C05472=1215.611,355.008,-74.397,-175.998,7.617,148.292
C05473=1215.607,355.256,-74.430,-175.997,7.621,148.293
C05474=1215.602,355.504,-74.463,-175.995,7.623,148.293
C05475=1215.599,355.752,-74.495,-175.993,7.626,148.293
C05476=1215.595,356.000,-74.528,-175.991,7.629,148.294
C05477=1215.590,356.248,-74.561,-175.990,7.632,148.294
C05478=1215.586,356.496,-74.594,-175.988,7.635,148.294
C05479=1215.582,356.743,-74.625,-175.986,7.638,148.294
C05480=1215.578,356.991,-74.658,-175.985,7.641,148.295
C05481=1215.573,357.239,-74.691,-175.983,7.644,148.295
C05482=1215.569,357.487,-74.724,-175.981,7.646,148.295
C05483=1215.566,357.734,-74.757,-175.979,7.649,148.295
C05484=1215.561,357.982,-74.789,-175.978,7.653,148.296
C05485=1215.557,358.230,-74.822,-175.976,7.655,148.296
C05486=1215.553,358.478,-74.855,-175.974,7.659,148.296
C05487=1215.549,358.726,-74.888,-175.973,7.661,148.297
C05488=1215.545,358.974,-74.920,-175.971,7.664,148.297
C05489=1215.541,359.221,-74.954,-175.969,7.667,148.297
C05490=1215.537,359.469,-74.987,-175.968,7.670,148.297
C05491=1215.533,359.718,-75.019,-175.966,7.673,148.298
C05492=1215.528,359.965,-75.052,-175.964,7.676,148.298
C05493=1215.524,360.212,-75.085,-175.963,7.679,148.298
C05494=1215.520,360.460,-75.118,-175.961,7.681,148.299
C05495=1215.516,360.708,-75.150,-175.959,7.685,148.299
C05496=1215.512,360.956,-75.183,-175.958,7.688,148.299
C05497=1215.508,361.203,-75.216,-175.956,7.690,148.299
C05498=1215.503,361.451,-75.250,-175.954,7.694,148.300
C05499=1215.499,361.699,-75.283,-175.953,7.696,148.300
C05500=1215.495,361.947,-75.316,-175.951,7.699,148.300
C05501=1215.491,362.195,-75.348,-175.950,7.703,148.301
C05502=1215.487,362.443,-75.381,-175.948,7.705,148.301
C05503=1215.482,362.690,-75.415,-175.947,7.708,148.301
C05504=1215.479,362.938,-75.447,-175.945,7.711,148.301
C05505=1215.475,363.186,-75.480,-175.943,7.714,148.302
C05506=1215.471,363.433,-75.513,-175.942,7.717,148.302
C05507=1215.467,363.681,-75.547,-175.941,7.719,148.302
C05508=1215.463,363.929,-75.580,-175.939,7.723,148.303
C05509=1215.458,364.177,-75.613,-175.937,7.726,148.303
C05510=1215.454,364.424,-75.646,-175.936,7.728,148.303
C05511=1215.450,364.673,-75.679,-175.934,7.732,148.304
C05512=1215.446,364.920,-75.712,-175.933,7.735,148.304
C05513=1215.442,365.168,-75.745,-175.931,7.737,148.304
C05514=1215.437,365.416,-75.778,-175.930,7.740,148.305
C05515=1215.433,365.664,-75.811,-175.928,7.744,148.305
C05516=1215.430,365.912,-75.845,-175.927,7.746,148.305
C05517=1215.426,366.160,-75.878,-175.925,7.749,148.306
C05518=1215.421,366.407,-75.911,-175.924,7.752,148.306
C05519=1215.417,366.687,-75.949,-175.922,7.755,148.306
C05520=1215.412,366.967,-75.986,-175.920,7.759,148.307
C05521=1215.408,367.247,-76.024,-175.919,7.761,148.307
C05522=1215.403,367.527,-76.061,-175.917,7.765,148.308
C05523=1215.398,367.775,-76.095,-175.916,7.768,148.308
C05524=1215.394,368.023,-76.128,-175.914,7.770,148.308
C05525=1215.390,368.270,-76.162,-175.913,7.773,148.309
C05526=1215.386,368.518,-76.195,-175.911,7.777,148.309
C05527=1215.382,368.765,-76.228,-175.910,7.780,148.309
C05528=1215.378,369.013,-76.261,-175.909,7.782,148.310
C05529=1215.374,369.261,-76.294,-175.907,7.785,148.310
C05530=1215.370,369.509,-76.328,-175.906,7.788,148.310
C05531=1215.366,369.757,-76.361,-175.905,7.792,148.311
C05532=1215.362,370.005,-76.394,-175.903,7.794,148.311
C05533=1215.358,370.252,-76.428,-175.902,7.797,148.311
C05534=1215.353,370.500,-76.462,-175.900,7.800,148.312
C05535=1215.349,370.748,-76.495,-175.899,7.803,148.312
C05536=1215.345,370.995,-76.528,-175.898,7.805,148.313
C05537=1215.341,371.243,-76.561,-175.897,7.808,148.313
C05538=1215.337,371.490,-76.595,-175.895,7.812,148.313
C05539=1215.334,371.739,-76.628,-175.894,7.814,148.314
C05540=1215.329,371.987,-76.662,-175.892,7.817,148.314
C05541=1215.325,372.234,-76.695,-175.891,7.820,148.314
C05542=1215.321,372.482,-76.729,-175.890,7.823,148.315
C05543=1215.317,372.729,-76.762,-175.889,7.826,148.315
C05544=1215.312,372.977,-76.796,-175.888,7.828,148.316
C05545=1215.308,373.225,-76.829,-175.886,7.831,148.316
C05546=1215.304,373.473,-76.864,-175.885,7.834,148.316
C05547=1215.300,373.721,-76.897,-175.884,7.837,148.317
C05548=1215.296,373.968,-76.930,-175.883,7.840,148.317
C05549=1215.292,374.215,-76.964,-175.881,7.843,148.318
C05550=1215.288,374.463,-76.997,-175.880,7.846,148.318
C05551=1215.283,374.711,-77.031,-175.879,7.849,148.318
C05552=1215.279,374.958,-77.065,-175.877,7.852,148.319
C05553=1215.276,375.207,-77.098,-175.876,7.855,148.319
C05554=1215.272,375.454,-77.131,-175.875,7.857,148.320
C05555=1215.268,375.702,-77.165,-175.874,7.860,148.320
C05556=1215.263,375.950,-77.199,-175.873,7.863,148.320
C05557=1215.259,376.197,-77.232,-175.872,7.866,148.321
C05558=1215.256,376.445,-77.266,-175.870,7.869,148.321
C05559=1215.252,376.693,-77.299,-175.869,7.871,148.322
C05560=1215.247,376.940,-77.334,-175.868,7.874,148.322
C05561=1215.243,377.188,-77.367,-175.867,7.877,148.322
C05562=1215.239,377.435,-77.401,-175.866,7.880,148.323
C05563=1215.235,377.684,-77.435,-175.864,7.883,148.323
C05564=1215.231,377.932,-77.468,-175.863,7.886,148.323
C05565=1215.227,378.179,-77.502,-175.862,7.888,148.324
C05566=1215.223,378.426,-77.535,-175.861,7.891,148.324
C05567=1215.218,378.674,-77.570,-175.860,7.894,148.325
C05568=1215.215,378.922,-77.603,-175.859,7.896,148.325
C05569=1215.211,379.169,-77.637,-175.858,7.899,148.326
C05570=1215.206,379.417,-77.671,-175.857,7.902,148.326
C05571=1215.202,379.665,-77.705,-175.856,7.905,148.326
C05572=1215.198,379.912,-77.738,-175.855,7.908,148.327
C05573=1215.194,380.160,-77.773,-175.853,7.910,148.327
C05574=1215.190,380.408,-77.806,-175.853,7.913,148.328
C05575=1215.186,380.655,-77.840,-175.852,7.916,148.328
C05576=1215.181,380.903,-77.873,-175.850,7.919,148.329
C05577=1215.178,381.151,-77.908,-175.849,7.922,148.329
C05578=1215.174,381.398,-77.942,-175.848,7.925,148.329
C05579=1215.169,381.646,-77.975,-175.848,7.927,148.330
C05580=1215.165,381.893,-78.009,-175.847,7.930,148.330
C05581=1215.161,382.142,-78.043,-175.845,7.933,148.331
C05582=1215.157,382.389,-78.077,-175.844,7.935,148.331
C05583=1215.153,382.636,-78.111,-175.843,7.939,148.332
C05584=1215.148,382.884,-78.145,-175.842,7.941,148.332
C05585=1215.145,383.132,-78.179,-175.842,7.943,148.332
C05586=1215.140,383.380,-78.213,-175.840,7.946,148.333
C05587=1215.137,383.627,-78.247,-175.840,7.949,148.333
C05588=1215.133,383.875,-78.281,-175.838,7.952,148.334
C05589=1215.128,384.123,-78.315,-175.837,7.955,148.334
C05590=1215.125,384.370,-78.348,-175.837,7.957,148.335
C05591=1215.120,384.618,-78.383,-175.836,7.960,148.335
C05592=1215.116,384.866,-78.416,-175.835,7.963,148.336
C05593=1215.112,385.114,-78.451,-175.834,7.966,148.336
C05594=1215.108,385.361,-78.485,-175.833,7.969,148.337
C05595=1215.105,385.608,-78.519,-175.832,7.971,148.337
C05596=1215.100,385.857,-78.553,-175.831,7.974,148.337
C05597=1215.096,386.104,-78.587,-175.830,7.977,148.338
C05598=1215.092,386.351,-78.621,-175.829,7.979,148.338
C05599=1215.088,386.599,-78.655,-175.828,7.981,148.339
C05600=1215.083,386.847,-78.689,-175.828,7.985,148.339
C05601=1215.080,387.094,-78.723,-175.826,7.987,148.340
C05602=1215.076,387.342,-78.758,-175.826,7.989,148.340
C05603=1215.072,387.590,-78.791,-175.825,7.992,148.340
C05604=1215.067,387.837,-78.825,-175.824,7.995,148.341
C05605=1215.064,388.085,-78.860,-175.824,7.998,148.341
C05606=1215.059,388.332,-78.894,-175.822,8.000,148.342
C05607=1215.055,388.580,-78.928,-175.821,8.003,148.342
C05608=1215.051,388.828,-78.962,-175.821,8.005,148.343
C05609=1215.047,389.075,-78.996,-175.820,8.008,148.343
C05610=1215.043,389.323,-79.030,-175.819,8.011,148.344
C05611=1215.039,389.571,-79.065,-175.818,8.013,148.344
C05612=1215.035,389.818,-79.099,-175.817,8.016,148.344
C05613=1215.031,390.066,-79.132,-175.817,8.019,148.345
C05614=1215.027,390.314,-79.167,-175.816,8.021,148.345
C05615=1215.023,390.561,-79.201,-175.815,8.024,148.346
C05616=1215.018,390.808,-79.235,-175.814,8.027,148.346
C05617=1215.015,391.056,-79.270,-175.814,8.029,148.347
C05618=1215.011,391.304,-79.304,-175.813,8.032,148.347
C05619=1215.007,391.552,-79.339,-175.812,8.035,148.348
C05620=1215.003,391.799,-79.373,-175.811,8.037,148.348
C05621=1214.998,392.047,-79.407,-175.811,8.039,148.349
C05622=1214.995,392.295,-79.441,-175.810,8.042,148.349
C05623=1214.990,392.576,-79.480,-175.809,8.046,148.350
C05624=1214.985,392.859,-79.519,-175.808,8.048,148.350
C05625=1214.981,393.141,-79.558,-175.807,8.051,148.351
C05626=1214.976,393.422,-79.598,-175.806,8.055,148.351
C05627=1214.972,393.670,-79.632,-175.806,8.057,148.352
C05628=1214.968,393.918,-79.666,-175.805,8.060,148.352
C05629=1214.963,394.166,-79.700,-175.804,8.062,148.353
C05630=1214.959,394.414,-79.735,-175.804,8.065,148.353
C05631=1214.956,394.661,-79.769,-175.803,8.067,148.354
C05632=1214.951,394.908,-79.803,-175.802,8.070,148.354
C05633=1214.948,395.156,-79.838,-175.802,8.072,148.355
C05634=1214.943,395.404,-79.872,-175.801,8.075,148.355
C05635=1214.939,395.652,-79.907,-175.800,8.077,148.355
C05636=1214.935,395.899,-79.941,-175.799,8.080,148.356
C05637=1214.931,396.146,-79.975,-175.799,8.082,148.356
C05638=1214.927,396.394,-80.010,-175.799,8.084,148.357
C05639=1214.923,396.641,-80.044,-175.797,8.087,148.357
C05640=1214.919,396.890,-80.079,-175.797,8.089,148.358
C05641=1214.915,397.137,-80.113,-175.796,8.092,148.358
C05642=1214.911,397.383,-80.148,-175.796,8.094,148.359
C05643=1214.907,397.632,-80.183,-175.795,8.097,148.359
C05644=1214.902,397.879,-80.217,-175.794,8.099,148.360
C05645=1214.899,398.127,-80.251,-175.794,8.101,148.360
C05646=1214.895,398.374,-80.286,-175.793,8.105,148.361
C05647=1214.891,398.622,-80.321,-175.792,8.107,148.361
C05648=1214.887,398.869,-80.355,-175.792,8.110,148.362
C05649=1214.882,399.117,-80.389,-175.791,8.112,148.362
C05650=1214.878,399.365,-80.424,-175.791,8.114,148.363
C05651=1214.875,399.612,-80.458,-175.790,8.117,148.363
C05652=1214.871,399.860,-80.493,-175.789,8.119,148.363
C05653=1214.866,400.108,-80.527,-175.789,8.121,148.364
C05654=1214.863,400.355,-80.562,-175.788,8.124,148.364
C05655=1214.858,400.602,-80.596,-175.788,8.126,148.365
C05656=1214.855,400.850,-80.631,-175.787,8.128,148.365
C05657=1214.850,401.098,-80.666,-175.786,8.131,148.366
C05658=1214.846,401.345,-80.700,-175.786,8.134,148.366
C05659=1214.842,401.593,-80.734,-175.785,8.136,148.367
C05660=1214.838,401.840,-80.769,-175.785,8.139,148.367
C05661=1214.834,402.088,-80.804,-175.784,8.141,148.368
C05662=1214.830,402.335,-80.838,-175.784,8.143,148.368
C05663=1214.826,402.583,-80.873,-175.783,8.145,148.369
C05664=1214.822,402.831,-80.908,-175.782,8.148,148.369
C05665=1214.818,403.079,-80.942,-175.782,8.150,148.369
C05666=1214.814,403.326,-80.976,-175.782,8.152,148.370
C05667=1214.810,403.573,-81.012,-175.781,8.155,148.371
C05668=1214.806,403.821,-81.046,-175.780,8.157,148.371
C05669=1214.802,404.069,-81.081,-175.780,8.160,148.371
C05670=1214.798,404.316,-81.115,-175.779,8.162,148.372
C05671=1214.794,404.563,-81.151,-175.779,8.165,148.372
C05672=1214.789,404.811,-81.185,-175.778,8.167,148.373
C05673=1214.786,405.059,-81.220,-175.778,8.169,148.373
C05674=1214.782,405.306,-81.254,-175.778,8.171,148.374
C05675=1214.778,405.554,-81.289,-175.777,8.173,148.374
C05676=1214.773,405.801,-81.324,-175.776,8.176,148.375
C05677=1214.769,406.049,-81.359,-175.775,8.178,148.375
C05678=1214.765,406.297,-81.393,-175.775,8.181,148.376
C05679=1214.762,406.544,-81.428,-175.775,8.183,148.376
C05680=1214.757,406.791,-81.462,-175.774,8.185,148.377
C05681=1214.753,407.039,-81.497,-175.774,8.188,148.377
C05682=1214.749,407.287,-81.532,-175.773,8.190,148.377
C05683=1214.745,407.534,-81.567,-175.773,8.192,148.378
C05684=1214.741,407.782,-81.602,-175.772,8.194,148.378
C05685=1214.737,408.029,-81.636,-175.772,8.196,148.379
C05686=1214.733,408.276,-81.671,-175.771,8.198,148.379
C05687=1214.729,408.524,-81.706,-175.771,8.202,148.380
C05688=1214.725,408.772,-81.741,-175.770,8.204,148.380
C05689=1214.721,409.019,-81.776,-175.770,8.206,148.381
C05690=1214.716,409.267,-81.811,-175.770,8.208,148.381
C05691=1214.713,409.514,-81.845,-175.769,8.210,148.382
C05692=1214.709,409.761,-81.880,-175.769,8.212,148.382
C05693=1214.705,410.009,-81.915,-175.768,8.214,148.382
C05694=1214.701,410.258,-81.950,-175.767,8.217,148.383
C05695=1214.697,410.504,-81.985,-175.767,8.219,148.383
C05696=1214.693,410.752,-82.020,-175.766,8.222,148.384
C05697=1214.689,411.000,-82.054,-175.766,8.224,148.384
C05698=1214.685,411.247,-82.089,-175.766,8.226,148.385
C05699=1214.681,411.494,-82.124,-175.765,8.228,148.385
C05700=1214.677,411.742,-82.159,-175.765,8.230,148.386
C05701=1214.672,411.989,-82.194,-175.764,8.232,148.386
C05702=1214.668,412.238,-82.228,-175.764,8.234,148.386
C05703=1214.664,412.484,-82.264,-175.764,8.237,148.387
C05704=1214.660,412.732,-82.298,-175.763,8.239,148.387
C05705=1214.657,412.980,-82.334,-175.763,8.241,148.388
C05706=1214.653,413.227,-82.368,-175.762,8.244,148.388
C05707=1214.649,413.475,-82.403,-175.761,8.246,148.389
C05708=1214.644,413.722,-82.438,-175.761,8.248,148.389
C05709=1214.641,413.970,-82.473,-175.761,8.250,148.390
C05710=1214.636,414.217,-82.508,-175.760,8.252,148.390
C05711=1214.632,414.465,-82.543,-175.760,8.254,148.391
C05712=1214.629,414.713,-82.578,-175.759,8.257,148.391
C05713=1214.624,414.960,-82.613,-175.759,8.259,148.391
C05714=1214.620,415.207,-82.648,-175.759,8.261,148.392
C05715=1214.616,415.442,-82.681,-175.758,8.263,148.392
C05716=1214.612,415.679,-82.714,-175.758,8.265,148.393
C05717=1214.608,415.914,-82.747,-175.757,8.267,148.393
C05718=1214.605,416.150,-82.781,-175.756,8.269,148.394
C05719=1214.601,416.385,-82.814,-175.757,8.271,148.394
C05720=1214.597,416.620,-82.848,-175.756,8.273,148.394
C05721=1214.595,416.856,-82.880,-175.756,8.275,148.395
C05722=1214.596,417.090,-82.914,-175.755,8.277,148.395
C05723=1214.175,417.091,-82.949,-175.759,8.287,148.399
C05724=1214.174,416.855,-82.917,-175.759,8.285,148.398
C05725=1214.175,416.618,-82.883,-175.759,8.283,148.398
C05726=1214.180,416.381,-82.849,-175.760,8.281,148.398
C05727=1214.183,416.144,-82.816,-175.760,8.280,148.397
C05728=1214.187,415.906,-82.782,-175.760,8.278,148.397
C05729=1214.190,415.671,-82.749,-175.761,8.276,148.396
C05730=1214.194,415.433,-82.715,-175.761,8.274,148.396
C05731=1214.199,415.197,-82.682,-175.761,8.271,148.396
C05732=1214.202,414.949,-82.647,-175.762,8.269,148.395
C05733=1214.206,414.702,-82.612,-175.762,8.267,148.395
C05734=1214.210,414.454,-82.577,-175.763,8.265,148.394
C05735=1214.215,414.207,-82.542,-175.763,8.263,148.394
C05736=1214.219,413.959,-82.507,-175.764,8.261,148.393
C05737=1214.222,413.711,-82.472,-175.764,8.259,148.393
C05738=1214.227,413.464,-82.437,-175.765,8.257,148.393
C05739=1214.230,413.217,-82.402,-175.765,8.254,148.392
C05740=1214.235,412.969,-82.367,-175.765,8.252,148.391
C05741=1214.239,412.721,-82.332,-175.766,8.249,148.391
C05742=1214.243,412.474,-82.297,-175.767,8.247,148.391
C05743=1214.247,412.226,-82.263,-175.767,8.245,148.390
C05744=1214.251,411.980,-82.228,-175.767,8.243,148.390
C05745=1214.255,411.731,-82.193,-175.768,8.241,148.389
C05746=1214.258,411.484,-82.157,-175.768,8.238,148.389
C05747=1214.263,411.237,-82.123,-175.769,8.236,148.388
C05748=1214.267,410.988,-82.088,-175.769,8.234,148.388
C05749=1214.271,410.742,-82.053,-175.769,8.232,148.387
C05750=1214.275,410.493,-82.018,-175.770,8.230,148.387
C05751=1214.279,410.246,-81.984,-175.770,8.228,148.387
C05752=1214.283,409.999,-81.949,-175.771,8.225,148.386
C05753=1214.287,409.751,-81.914,-175.772,8.223,148.386
C05754=1214.291,409.504,-81.879,-175.772,8.221,148.385
C05755=1214.295,409.257,-81.844,-175.772,8.218,148.385
C05756=1214.299,409.008,-81.809,-175.773,8.216,148.384
C05757=1214.303,408.761,-81.774,-175.773,8.214,148.384
C05758=1214.307,408.514,-81.740,-175.774,8.212,148.383
C05759=1214.311,408.266,-81.705,-175.774,8.210,148.383
C05760=1214.315,408.019,-81.670,-175.775,8.207,148.382
C05761=1214.319,407.771,-81.635,-175.776,8.205,148.382
C05762=1214.324,407.523,-81.601,-175.776,8.203,148.382
C05763=1214.327,407.276,-81.565,-175.776,8.200,148.381
C05764=1214.331,407.029,-81.531,-175.777,8.198,148.381
C05765=1214.335,406.781,-81.496,-175.777,8.196,148.380
C05766=1214.340,406.533,-81.462,-175.778,8.193,148.380
C05767=1214.343,406.286,-81.426,-175.778,8.191,148.379
C05768=1214.348,406.038,-81.392,-175.779,8.189,148.379
C05769=1214.351,405.790,-81.358,-175.779,8.187,148.378
C05770=1214.355,405.544,-81.323,-175.779,8.184,148.378
C05771=1214.359,405.296,-81.288,-175.780,8.182,148.377
C05772=1214.364,405.048,-81.253,-175.781,8.179,148.377
C05773=1214.368,404.800,-81.218,-175.781,8.177,148.377
C05774=1214.372,404.554,-81.184,-175.782,8.175,148.376
C05775=1214.375,404.305,-81.149,-175.783,8.172,148.376
C05776=1214.380,404.058,-81.115,-175.783,8.170,148.375
C05777=1214.384,403.810,-81.080,-175.783,8.168,148.374
C05778=1214.388,403.563,-81.046,-175.784,8.166,148.374
C05779=1214.392,403.315,-81.010,-175.785,8.163,148.374
C05780=1214.396,403.068,-80.976,-175.785,8.161,148.373
C05781=1214.400,402.820,-80.941,-175.785,8.158,148.373
C05782=1214.405,402.572,-80.907,-175.786,8.156,148.372
C05783=1214.408,402.324,-80.872,-175.787,8.153,148.372
C05784=1214.412,402.078,-80.837,-175.787,8.151,148.371
C05785=1214.416,401.830,-80.802,-175.788,8.149,148.371
C05786=1214.421,401.582,-80.768,-175.788,8.146,148.370
C05787=1214.424,401.334,-80.734,-175.789,8.144,148.370
C05788=1214.428,401.087,-80.699,-175.789,8.142,148.369
C05789=1214.433,400.840,-80.665,-175.790,8.139,148.369
C05790=1214.436,400.592,-80.630,-175.791,8.137,148.368
C05791=1214.441,400.345,-80.595,-175.791,8.134,148.368
C05792=1214.444,400.097,-80.560,-175.792,8.132,148.368
C05793=1214.449,399.849,-80.526,-175.792,8.129,148.367
C05794=1214.452,399.602,-80.492,-175.793,8.127,148.367
C05795=1214.457,399.354,-80.457,-175.794,8.124,148.366
C05796=1214.461,399.106,-80.422,-175.794,8.122,148.366
C05797=1214.465,398.859,-80.389,-175.795,8.120,148.365
C05798=1214.469,398.612,-80.353,-175.796,8.117,148.365
C05799=1214.473,398.364,-80.318,-175.796,8.115,148.364
C05800=1214.477,398.117,-80.285,-175.796,8.113,148.364
C05801=1214.481,397.869,-80.250,-175.797,8.110,148.363
C05802=1214.485,397.621,-80.215,-175.797,8.108,148.363
C05803=1214.489,397.373,-80.180,-175.799,8.105,148.362
C05804=1214.493,397.126,-80.147,-175.799,8.102,148.362
C05805=1214.498,396.879,-80.112,-175.800,8.100,148.361
C05806=1214.502,396.631,-80.077,-175.800,8.097,148.361
C05807=1214.505,396.383,-80.043,-175.801,8.095,148.361
C05808=1214.509,396.135,-80.009,-175.802,8.092,148.360
C05809=1214.513,395.888,-79.975,-175.802,8.090,148.360
C05810=1214.517,395.640,-79.940,-175.803,8.087,148.359
C05811=1214.522,395.393,-79.905,-175.804,8.085,148.359
C05812=1214.526,395.146,-79.872,-175.804,8.082,148.358
C05813=1214.530,394.897,-79.837,-175.805,8.080,148.358
C05814=1214.534,394.650,-79.802,-175.806,8.077,148.357
C05815=1214.537,394.402,-79.768,-175.806,8.075,148.357
C05816=1214.542,394.155,-79.734,-175.807,8.072,148.356
C05817=1214.546,393.908,-79.700,-175.807,8.070,148.356
C05818=1214.550,393.660,-79.665,-175.809,8.067,148.355
C05819=1214.554,393.412,-79.630,-175.809,8.065,148.355
C05820=1214.558,393.130,-79.591,-175.810,8.062,148.354
C05821=1214.563,392.848,-79.552,-175.811,8.059,148.354
C05822=1214.568,392.566,-79.513,-175.812,8.056,148.353
C05823=1214.573,392.283,-79.474,-175.813,8.053,148.353
C05824=1214.576,392.036,-79.440,-175.813,8.050,148.352
C05825=1214.581,391.789,-79.406,-175.814,8.048,148.352
C05826=1214.584,391.541,-79.371,-175.815,8.045,148.351
C05827=1214.589,391.293,-79.337,-175.816,8.043,148.351
C05828=1214.593,391.046,-79.303,-175.816,8.039,148.350
C05829=1214.597,390.798,-79.268,-175.817,8.038,148.350
C05830=1214.601,390.550,-79.234,-175.818,8.034,148.349
C05831=1214.605,390.302,-79.200,-175.819,8.032,148.349
C05832=1214.609,390.055,-79.166,-175.820,8.030,148.349
C05833=1214.613,389.808,-79.132,-175.820,8.026,148.348
C05834=1214.617,389.560,-79.097,-175.821,8.025,148.348
C05835=1214.621,389.313,-79.063,-175.822,8.021,148.347
C05836=1214.625,389.065,-79.029,-175.823,8.019,148.347
C05837=1214.629,388.817,-78.995,-175.823,8.016,148.346
C05838=1214.633,388.569,-78.961,-175.824,8.014,148.346
C05839=1214.637,388.322,-78.927,-175.825,8.011,148.345
C05840=1214.641,388.074,-78.892,-175.826,8.008,148.345
C05841=1214.645,387.827,-78.858,-175.827,8.006,148.344
C05842=1214.650,387.579,-78.824,-175.828,8.003,148.344
C05843=1214.653,387.331,-78.790,-175.828,8.001,148.344
C05844=1214.658,387.084,-78.756,-175.829,7.998,148.343
C05845=1214.662,386.837,-78.722,-175.830,7.995,148.343
C05846=1214.666,386.588,-78.688,-175.831,7.992,148.342
C05847=1214.670,386.341,-78.654,-175.832,7.990,148.342
C05848=1214.674,386.093,-78.619,-175.833,7.987,148.341
C05849=1214.678,385.846,-78.585,-175.834,7.984,148.341
C05850=1214.682,385.598,-78.551,-175.835,7.981,148.340
C05851=1214.686,385.350,-78.517,-175.835,7.979,148.340
C05852=1214.691,385.103,-78.483,-175.837,7.976,148.339
C05853=1214.694,384.855,-78.449,-175.838,7.973,148.339
C05854=1214.698,384.607,-78.416,-175.838,7.970,148.338
C05855=1214.703,384.360,-78.381,-175.839,7.968,148.338
C05856=1214.706,384.112,-78.347,-175.840,7.965,148.338
C05857=1214.711,383.864,-78.313,-175.841,7.962,148.337
C05858=1214.715,383.617,-78.279,-175.842,7.959,148.337
C05859=1214.719,383.370,-78.245,-175.843,7.957,148.336
C05860=1214.723,383.121,-78.211,-175.844,7.955,148.336
C05861=1214.727,382.874,-78.177,-175.845,7.951,148.335
C05862=1214.732,382.626,-78.144,-175.846,7.949,148.335
C05863=1214.735,382.378,-78.109,-175.847,7.946,148.335
C05864=1214.739,382.131,-78.075,-175.848,7.943,148.334
C05865=1214.743,381.883,-78.042,-175.849,7.940,148.334
C05866=1214.747,381.636,-78.008,-175.850,7.937,148.333
C05867=1214.752,381.387,-77.974,-175.851,7.935,148.333
C05868=1214.755,381.140,-77.940,-175.852,7.932,148.333
C05869=1214.759,380.893,-77.906,-175.853,7.929,148.332
C05870=1214.764,380.645,-77.872,-175.854,7.926,148.332
C05871=1214.767,380.397,-77.838,-175.855,7.924,148.331
C05872=1214.772,380.149,-77.804,-175.856,7.921,148.331
C05873=1214.776,379.902,-77.770,-175.858,7.918,148.330
C05874=1214.780,379.654,-77.737,-175.858,7.915,148.330
C05875=1214.785,379.407,-77.703,-175.860,7.912,148.329
C05876=1214.788,379.158,-77.669,-175.861,7.909,148.329
C05877=1214.792,378.911,-77.635,-175.861,7.907,148.329
C05878=1214.797,378.663,-77.602,-175.863,7.904,148.328
C05879=1214.801,378.416,-77.568,-175.864,7.902,148.328
C05880=1214.804,378.168,-77.534,-175.865,7.899,148.327
C05881=1214.808,377.921,-77.500,-175.866,7.896,148.327
C05882=1214.813,377.673,-77.467,-175.867,7.893,148.326
C05883=1214.817,377.426,-77.433,-175.868,7.890,148.326
C05884=1214.821,377.178,-77.400,-175.869,7.887,148.326
C05885=1214.825,376.930,-77.365,-175.871,7.884,148.325
C05886=1214.829,376.682,-77.332,-175.872,7.882,148.325
C05887=1214.833,376.434,-77.298,-175.873,7.879,148.324
C05888=1214.837,376.187,-77.265,-175.874,7.876,148.324
C05889=1214.842,375.939,-77.231,-175.875,7.873,148.324
C05890=1214.845,375.691,-77.197,-175.876,7.870,148.323
C05891=1214.849,375.444,-77.163,-175.878,7.867,148.323
C05892=1214.853,375.196,-77.130,-175.879,7.865,148.323
C05893=1214.858,374.948,-77.096,-175.880,7.862,148.322
C05894=1214.862,374.701,-77.063,-175.881,7.859,148.322
C05895=1214.866,374.453,-77.030,-175.882,7.856,148.321
C05896=1214.870,374.205,-76.995,-175.884,7.853,148.321
C05897=1214.874,373.957,-76.962,-175.885,7.850,148.320
C05898=1214.879,373.709,-76.928,-175.887,7.847,148.320
C05899=1214.882,373.462,-76.895,-175.888,7.844,148.320
C05900=1214.887,373.215,-76.861,-175.889,7.841,148.319
C05901=1214.891,372.967,-76.828,-175.890,7.839,148.319
C05902=1214.895,372.720,-76.794,-175.891,7.836,148.319
C05903=1214.899,372.471,-76.760,-175.893,7.833,148.318
C05904=1214.903,372.223,-76.727,-175.894,7.830,148.318
C05905=1214.907,371.975,-76.694,-175.895,7.827,148.317
C05906=1214.911,371.728,-76.660,-175.897,7.825,148.317
C05907=1214.915,371.481,-76.627,-175.898,7.821,148.317
C05908=1214.919,371.233,-76.594,-175.900,7.818,148.316
C05909=1214.923,370.985,-76.561,-175.901,7.815,148.316
C05910=1214.927,370.737,-76.526,-175.902,7.813,148.316
C05911=1214.931,370.489,-76.493,-175.903,7.810,148.315
C05912=1214.936,370.242,-76.459,-175.904,7.807,148.315
C05913=1214.940,369.994,-76.426,-175.906,7.804,148.315
C05914=1214.944,369.746,-76.393,-175.908,7.801,148.314
C05915=1214.948,369.498,-76.360,-175.909,7.798,148.314
C05916=1214.952,369.251,-76.326,-175.910,7.795,148.313
C05917=1214.956,369.004,-76.293,-175.911,7.792,148.313
C05918=1214.960,368.756,-76.260,-175.913,7.790,148.313
C05919=1214.965,368.508,-76.226,-175.915,7.786,148.312
C05920=1214.969,368.260,-76.193,-175.916,7.783,148.312
C05921=1214.973,368.012,-76.159,-175.917,7.781,148.312
C05922=1214.977,367.764,-76.126,-175.919,7.778,148.311
C05923=1214.981,367.516,-76.093,-175.920,7.775,148.311
C05924=1214.986,367.237,-76.056,-175.922,7.772,148.311
C05925=1214.990,366.957,-76.018,-175.923,7.768,148.310
C05926=1214.994,366.677,-75.980,-175.925,7.765,148.310
C05927=1215.000,366.396,-75.943,-175.927,7.762,148.309
C05928=1215.004,366.148,-75.910,-175.928,7.759,148.309
C05929=1215.008,365.901,-75.876,-175.930,7.756,148.309
C05930=1215.012,365.653,-75.843,-175.931,7.753,148.308
C05931=1215.016,365.405,-75.810,-175.932,7.750,148.308
C05932=1215.020,365.158,-75.777,-175.934,7.747,148.308
C05933=1215.025,364.910,-75.744,-175.936,7.744,148.307
C05934=1215.029,364.662,-75.711,-175.937,7.741,148.307
C05935=1215.033,364.414,-75.677,-175.939,7.738,148.307
C05936=1215.037,364.167,-75.644,-175.940,7.736,148.306
C05937=1215.040,363.919,-75.612,-175.942,7.732,148.306
C05938=1215.044,363.671,-75.578,-175.943,7.729,148.306
C05939=1215.048,363.423,-75.545,-175.944,7.727,148.305
C05940=1215.052,363.175,-75.512,-175.947,7.723,148.305
C05941=1215.056,362.928,-75.479,-175.948,7.720,148.305
C05942=1215.060,362.680,-75.446,-175.949,7.718,148.305
C05943=1215.065,362.432,-75.412,-175.951,7.715,148.304
C05944=1215.069,362.184,-75.380,-175.953,7.712,148.304
C05945=1215.073,361.936,-75.347,-175.954,7.709,148.304
C05946=1215.077,361.688,-75.314,-175.956,7.706,148.303
C05947=1215.082,361.441,-75.281,-175.957,7.703,148.303
C05948=1215.086,361.194,-75.248,-175.959,7.700,148.303
C05949=1215.090,360.946,-75.215,-175.960,7.697,148.302
C05950=1215.094,360.698,-75.183,-175.962,7.694,148.302
C05951=1215.098,360.450,-75.150,-175.964,7.692,148.302
C05952=1215.102,360.202,-75.116,-175.965,7.689,148.302
C05953=1215.106,359.955,-75.083,-175.967,7.685,148.301
C05954=1215.111,359.707,-75.050,-175.969,7.683,148.301
C05955=1215.115,359.459,-75.018,-175.970,7.680,148.301
C05956=1215.118,359.211,-74.985,-175.973,7.677,148.300
C05957=1215.123,358.963,-74.952,-175.974,7.674,148.300
C05958=1215.127,358.715,-74.919,-175.976,7.671,148.300
C05959=1215.131,358.467,-74.886,-175.977,7.668,148.299
C05960=1215.135,358.220,-74.853,-175.979,7.665,148.299
C05961=1215.139,357.972,-74.820,-175.981,7.662,148.299
C05962=1215.143,357.724,-74.788,-175.982,7.659,148.299
C05963=1215.147,357.476,-74.755,-175.984,7.657,148.298
C05964=1215.151,357.228,-74.722,-175.986,7.653,148.298
C05965=1215.156,356.980,-74.689,-175.987,7.650,148.298
C05966=1215.160,356.733,-74.657,-175.989,7.647,148.298
C05967=1215.164,356.486,-74.624,-175.991,7.644,148.297
C05968=1215.168,356.237,-74.592,-175.992,7.642,148.297
C05969=1215.173,355.989,-74.558,-175.994,7.638,148.297
C05970=1215.176,355.741,-74.527,-175.996,7.636,148.297
C05971=1215.180,355.494,-74.493,-175.998,7.633,148.296
C05972=1215.185,355.246,-74.460,-175.999,7.630,148.296
C05973=1215.189,354.998,-74.428,-176.001,7.627,148.296
C05974=1215.192,354.750,-74.395,-176.003,7.624,148.296
C05975=1215.197,354.503,-74.363,-176.005,7.621,148.295
C05976=1215.202,354.255,-74.330,-176.007,7.619,148.295
C05977=1215.206,354.007,-74.298,-176.008,7.615,148.295
C05978=1215.209,353.759,-74.265,-176.010,7.613,148.295
C05979=1215.214,353.511,-74.233,-176.012,7.609,148.294
C05980=1215.218,353.263,-74.199,-176.014,7.607,148.294
C05981=1215.222,353.016,-74.168,-176.016,7.603,148.294
C05982=1215.226,352.768,-74.135,-176.017,7.601,148.294
C05983=1215.231,352.520,-74.102,-176.019,7.598,148.293
C05984=1215.234,352.272,-74.070,-176.021,7.595,148.293
C05985=1215.239,352.024,-74.037,-176.023,7.592,148.293
C05986=1215.243,351.775,-74.005,-176.025,7.589,148.293
C05987=1215.247,351.529,-73.973,-176.026,7.586,148.293
C05988=1215.252,351.280,-73.940,-176.028,7.584,148.292
C05989=1215.255,351.033,-73.908,-176.030,7.580,148.292
C05990=1215.260,350.785,-73.875,-176.032,7.578,148.292
C05991=1215.264,350.536,-73.843,-176.034,7.574,148.292
C05992=1215.268,350.290,-73.811,-176.035,7.572,148.291
C05993=1215.272,350.041,-73.778,-176.038,7.568,148.291
C05994=1215.276,349.793,-73.746,-176.039,7.566,148.291
C05995=1215.280,349.545,-73.713,-176.041,7.563,148.291
C05996=1215.285,349.297,-73.681,-176.043,7.560,148.291
C05997=1215.289,349.050,-73.649,-176.045,7.557,148.290
C05998=1215.293,348.802,-73.616,-176.047,7.554,148.290
C05999=1215.297,348.554,-73.584,-176.049,7.552,148.290
C06000=1215.301,348.306,-73.552,-176.051,7.548,148.290
C06001=1215.306,348.058,-73.520,-176.052,7.546,148.290
C06002=1215.310,347.811,-73.487,-176.054,7.543,148.289
C06003=1215.313,347.563,-73.455,-176.056,7.540,148.289
C06004=1215.318,347.314,-73.423,-176.058,7.537,148.289
C06005=1215.322,347.067,-73.392,-176.060,7.534,148.289
C06006=1215.326,346.819,-73.358,-176.062,7.531,148.289
C06007=1215.330,346.571,-73.327,-176.064,7.528,148.288
C06008=1215.334,346.323,-73.294,-176.066,7.526,148.288
C06009=1215.339,346.075,-73.263,-176.068,7.522,148.288
C06010=1215.343,345.827,-73.230,-176.069,7.520,148.288
C06011=1215.347,345.579,-73.198,-176.071,7.517,148.288
C06012=1215.351,345.331,-73.165,-176.073,7.514,148.287
C06013=1215.355,345.084,-73.134,-176.075,7.511,148.287
C06014=1215.360,344.836,-73.101,-176.077,7.508,148.287
C06015=1215.364,344.588,-73.069,-176.079,7.505,148.287
C06016=1215.369,344.340,-73.037,-176.081,7.502,148.287
C06017=1215.372,344.092,-73.005,-176.083,7.500,148.286
C06018=1215.376,343.844,-72.974,-176.085,7.496,148.286
C06019=1215.381,343.596,-72.942,-176.087,7.494,148.286
C06020=1215.385,343.348,-72.910,-176.089,7.491,148.286
C06021=1215.389,343.100,-72.877,-176.091,7.488,148.286
C06022=1215.393,342.852,-72.846,-176.092,7.486,148.286
C06023=1215.397,342.604,-72.814,-176.095,7.482,148.285
C06024=1215.402,342.356,-72.781,-176.096,7.480,148.285
C06025=1215.406,342.109,-72.750,-176.099,7.477,148.285
C06026=1215.410,341.860,-72.718,-176.101,7.474,148.285
C06027=1215.414,341.612,-72.686,-176.103,7.471,148.285
C06028=1215.418,341.335,-72.650,-176.105,7.467,148.285
C06029=1215.423,341.057,-72.614,-176.107,7.464,148.284
C06030=1215.428,340.779,-72.579,-176.109,7.462,148.284
C06031=1215.433,340.501,-72.543,-176.111,7.459,148.284
C06032=1215.437,340.253,-72.511,-176.114,7.455,148.284
C06033=1215.441,340.006,-72.479,-176.115,7.453,148.284
C06034=1215.446,339.757,-72.447,-176.117,7.449,148.283
C06035=1215.449,339.509,-72.415,-176.120,7.447,148.284
C06036=1215.454,339.261,-72.384,-176.122,7.444,148.283
C06037=1215.458,339.013,-72.352,-176.123,7.441,148.283
C06038=1215.463,338.766,-72.321,-176.126,7.438,148.283
C06039=1215.466,338.518,-72.289,-176.128,7.436,148.283
C06040=1215.470,338.269,-72.257,-176.130,7.432,148.283
C06041=1215.475,338.022,-72.225,-176.132,7.430,148.283
C06042=1215.479,337.773,-72.194,-176.134,7.427,148.283
C06043=1215.483,337.526,-72.162,-176.136,7.424,148.282
C06044=1215.487,337.278,-72.130,-176.138,7.421,148.282
C06045=1215.492,337.029,-72.098,-176.140,7.418,148.282
C06046=1215.496,336.782,-72.066,-176.142,7.415,148.282
C06047=1215.500,336.533,-72.035,-176.144,7.413,148.282
C06048=1215.504,336.286,-72.004,-176.146,7.409,148.282
C06049=1215.508,336.038,-71.972,-176.148,7.407,148.282
C06050=1215.513,335.790,-71.941,-176.150,7.405,148.281
C06051=1215.517,335.542,-71.909,-176.152,7.401,148.281
C06052=1215.521,335.294,-71.877,-176.154,7.399,148.281
C06053=1215.525,335.046,-71.846,-176.156,7.396,148.281
C06054=1215.529,334.798,-71.814,-176.158,7.393,148.281
C06055=1215.533,334.550,-71.783,-176.161,7.390,148.281
C06056=1215.537,334.302,-71.752,-176.162,7.388,148.281
C06057=1215.542,334.054,-71.720,-176.165,7.385,148.281
C06058=1215.546,333.806,-71.688,-176.167,7.382,148.280
C06059=1215.551,333.558,-71.657,-176.169,7.379,148.280
C06060=1215.554,333.310,-71.625,-176.171,7.377,148.280
C06061=1215.559,333.062,-71.594,-176.173,7.373,148.280
C06062=1215.563,332.814,-71.563,-176.175,7.371,148.280
C06063=1215.567,332.567,-71.531,-176.178,7.368,148.280
C06064=1215.571,332.318,-71.500,-176.179,7.365,148.280
C06065=1215.575,332.071,-71.468,-176.182,7.362,148.280
C06066=1215.579,331.822,-71.437,-176.184,7.360,148.280
C06067=1215.584,331.575,-71.406,-176.186,7.356,148.280
C06068=1215.588,331.326,-71.375,-176.188,7.354,148.279
C06069=1215.593,331.078,-71.343,-176.190,7.351,148.279
C06070=1215.597,330.830,-71.311,-176.192,7.348,148.279
C06071=1215.601,330.582,-71.280,-176.195,7.345,148.279
C06072=1215.606,330.334,-71.249,-176.196,7.343,148.279
C06073=1215.610,330.086,-71.218,-176.199,7.340,148.279
C06074=1215.614,329.838,-71.187,-176.201,7.337,148.279
C06075=1215.618,329.590,-71.156,-176.203,7.334,148.279
C06076=1215.622,329.342,-71.124,-176.205,7.332,148.279
C06077=1215.626,329.094,-71.093,-176.208,7.329,148.279
C06078=1215.631,328.846,-71.062,-176.209,7.326,148.278
C06079=1215.635,328.599,-71.031,-176.212,7.323,148.278
C06080=1215.639,328.350,-71.000,-176.214,7.321,148.278
C06081=1215.643,328.103,-70.969,-176.216,7.318,148.278
C06082=1215.647,327.854,-70.938,-176.218,7.315,148.278
C06083=1215.651,327.606,-70.907,-176.221,7.312,148.278
C06084=1215.655,327.358,-70.876,-176.222,7.309,148.278
C06085=1215.660,327.110,-70.844,-176.225,7.306,148.278
C06086=1215.664,326.862,-70.813,-176.227,7.304,148.278
C06087=1215.668,326.614,-70.782,-176.229,7.301,148.278
C06088=1215.673,326.366,-70.751,-176.231,7.299,148.278
C06089=1215.677,326.118,-70.720,-176.234,7.295,148.278
C06090=1215.681,325.870,-70.689,-176.236,7.293,148.278
C06091=1215.685,325.622,-70.659,-176.238,7.290,148.277
C06092=1215.689,325.374,-70.627,-176.240,7.287,148.277
C06093=1215.694,325.126,-70.596,-176.243,7.284,148.277
C06094=1215.698,324.878,-70.565,-176.244,7.282,148.277
C06095=1215.702,324.629,-70.534,-176.247,7.279,148.277
C06096=1215.707,324.381,-70.503,-176.249,7.276,148.277
C06097=1215.711,324.133,-70.473,-176.251,7.273,148.277
C06098=1215.714,323.886,-70.441,-176.253,7.271,148.277
C06099=1215.719,323.638,-70.411,-176.256,7.268,148.277
C06100=1215.724,323.390,-70.380,-176.258,7.266,148.277
C06101=1215.728,323.141,-70.349,-176.260,7.262,148.277
C06102=1215.732,322.893,-70.318,-176.262,7.260,148.277
C06103=1215.736,322.646,-70.288,-176.265,7.257,148.277
C06104=1215.740,322.397,-70.257,-176.266,7.254,148.277
C06105=1215.745,322.149,-70.226,-176.268,7.252,148.277
C06106=1215.749,321.901,-70.195,-176.271,7.249,148.277
C06107=1215.753,321.653,-70.165,-176.273,7.247,148.277
C06108=1215.757,321.405,-70.133,-176.275,7.244,148.276
C06109=1215.762,321.157,-70.102,-176.278,7.241,148.277
C06110=1215.766,320.909,-70.071,-176.280,7.238,148.277
C06111=1215.769,320.661,-70.041,-176.282,7.236,148.276
C06112=1215.774,320.413,-70.010,-176.285,7.233,148.276
C06113=1215.779,320.165,-69.980,-176.287,7.231,148.276
C06114=1215.782,319.916,-69.950,-176.289,7.227,148.276
C06115=1215.787,319.668,-69.919,-176.291,7.225,148.276
C06116=1215.791,319.420,-69.888,-176.294,7.222,148.276
C06117=1215.795,319.172,-69.858,-176.296,7.220,148.276
C06118=1215.799,318.924,-69.827,-176.298,7.216,148.276
C06119=1215.804,318.676,-69.796,-176.300,7.214,148.276
C06120=1215.808,318.428,-69.766,-176.303,7.211,148.276
C06121=1215.812,318.180,-69.735,-176.305,7.209,148.276
C06122=1215.816,317.932,-69.704,-176.307,7.206,148.276
C06123=1215.820,317.684,-69.674,-176.309,7.203,148.276
C06124=1215.825,317.435,-69.644,-176.312,7.200,148.276
C06125=1215.830,317.188,-69.613,-176.314,7.198,148.276
C06126=1215.833,316.939,-69.583,-176.316,7.195,148.276
C06127=1215.838,316.691,-69.552,-176.318,7.193,148.276
C06128=1215.842,316.444,-69.522,-176.321,7.189,148.276
C06129=1215.847,316.195,-69.492,-176.323,7.187,148.276
C06130=1215.851,315.947,-69.461,-176.326,7.184,148.276
C06131=1215.854,315.699,-69.430,-176.327,7.182,148.276
C06132=1215.859,315.423,-69.396,-176.330,7.179,148.276
C06133=1215.864,315.146,-69.362,-176.333,7.176,148.276
C06134=1215.868,314.871,-69.329,-176.335,7.173,148.276
C06135=1215.874,314.595,-69.296,-176.338,7.170,148.276
C06136=1215.878,314.347,-69.264,-176.340,7.167,148.276
C06137=1215.882,314.099,-69.234,-176.343,7.164,148.276
C06138=1215.887,313.850,-69.204,-176.345,7.162,148.276
C06139=1215.891,313.603,-69.174,-176.347,7.159,148.276
C06140=1215.895,313.355,-69.143,-176.349,7.157,148.276
C06141=1215.899,313.107,-69.114,-176.352,7.153,148.276
C06142=1215.903,312.858,-69.083,-176.354,7.151,148.276
C06143=1215.908,312.610,-69.053,-176.357,7.148,148.276
C06144=1215.912,312.362,-69.023,-176.359,7.146,148.276
C06145=1215.916,312.114,-68.992,-176.361,7.144,148.276
C06146=1215.921,311.865,-68.962,-176.363,7.140,148.276
C06147=1215.925,311.618,-68.932,-176.365,7.138,148.276
C06148=1215.929,311.370,-68.903,-176.368,7.135,148.276
C06149=1215.934,311.122,-68.872,-176.370,7.133,148.276
C06150=1215.937,310.873,-68.842,-176.373,7.130,148.276
C06151=1215.942,310.625,-68.811,-176.375,7.128,148.276
C06152=1215.946,310.376,-68.782,-176.377,7.125,148.276
C06153=1215.951,310.128,-68.751,-176.380,7.122,148.276
C06154=1215.955,309.880,-68.722,-176.382,7.119,148.276
C06155=1215.959,309.632,-68.691,-176.384,7.117,148.276
C06156=1215.964,309.384,-68.661,-176.387,7.114,148.276
C06157=1215.968,309.136,-68.631,-176.389,7.112,148.276
C06158=1215.972,308.888,-68.602,-176.391,7.109,148.276
C06159=1215.976,308.640,-68.571,-176.393,7.106,148.276
C06160=1215.981,308.392,-68.542,-176.396,7.103,148.276
C06161=1215.985,308.143,-68.512,-176.398,7.101,148.276
C06162=1215.989,307.896,-68.481,-176.400,7.099,148.276
C06163=1215.994,307.647,-68.452,-176.403,7.096,148.276
C06164=1215.998,307.399,-68.421,-176.405,7.094,148.276
C06165=1216.002,307.151,-68.392,-176.408,7.091,148.276
C06166=1216.007,306.903,-68.362,-176.410,7.088,148.276
C06167=1216.010,306.654,-68.332,-176.413,7.085,148.276
C06168=1216.015,306.406,-68.302,-176.415,7.083,148.276
C06169=1216.019,306.158,-68.272,-176.417,7.080,148.276
C06170=1216.023,305.910,-68.242,-176.420,7.078,148.276
C06171=1216.028,305.661,-68.212,-176.422,7.075,148.276
C06172=1216.032,305.413,-68.183,-176.424,7.073,148.276
C06173=1216.036,305.165,-68.153,-176.427,7.070,148.276
C06174=1216.040,304.917,-68.123,-176.429,7.067,148.276
C06175=1216.045,304.669,-68.093,-176.431,7.065,148.276
C06176=1216.050,304.421,-68.064,-176.434,7.062,148.276
C06177=1216.054,304.173,-68.034,-176.436,7.060,148.276
C06178=1216.058,303.925,-68.005,-176.439,7.057,148.276
C06179=1216.063,303.677,-67.974,-176.441,7.055,148.277
C06180=1216.067,303.428,-67.945,-176.443,7.052,148.277
C06181=1216.071,303.180,-67.915,-176.446,7.050,148.277
C06182=1216.075,302.932,-67.886,-176.448,7.046,148.277
C06183=1216.079,302.683,-67.856,-176.450,7.044,148.277
C06184=1216.084,302.435,-67.827,-176.452,7.042,148.277
C06185=1216.088,302.187,-67.797,-176.455,7.039,148.277
C06186=1216.092,301.939,-67.767,-176.457,7.037,148.277
C06187=1216.096,301.691,-67.737,-176.460,7.034,148.277
C06188=1216.101,301.442,-67.708,-176.462,7.032,148.277
C06189=1216.105,301.194,-67.678,-176.465,7.029,148.277
C06190=1216.109,300.946,-67.649,-176.467,7.026,148.277
C06191=1216.113,300.698,-67.619,-176.470,7.024,148.277
C06192=1216.117,300.449,-67.590,-176.472,7.021,148.277
C06193=1216.123,300.202,-67.560,-176.474,7.019,148.277
C06194=1216.127,299.953,-67.531,-176.477,7.016,148.277
C06195=1216.131,299.705,-67.501,-176.479,7.014,148.277
C06196=1216.135,299.457,-67.472,-176.482,7.011,148.277
C06197=1216.140,299.208,-67.442,-176.484,7.009,148.277
C06198=1216.144,298.960,-67.413,-176.486,7.006,148.277
C06199=1216.148,298.712,-67.384,-176.489,7.003,148.278
C06200=1216.152,298.464,-67.354,-176.491,7.001,148.278
C06201=1216.156,298.215,-67.325,-176.494,6.999,148.278
C06202=1216.161,297.968,-67.296,-176.496,6.996,148.278
C06203=1216.165,297.720,-67.266,-176.499,6.993,148.278
C06204=1216.170,297.471,-67.237,-176.501,6.991,148.278
C06205=1216.174,297.222,-67.208,-176.503,6.988,148.278
C06206=1216.178,296.974,-67.178,-176.506,6.986,148.278
C06207=1216.182,296.726,-67.149,-176.508,6.984,148.278
C06208=1216.187,296.478,-67.120,-176.510,6.981,148.278
C06209=1216.191,296.230,-67.090,-176.513,6.979,148.278
C06210=1216.196,295.982,-67.061,-176.516,6.976,148.278
C06211=1216.200,295.733,-67.032,-176.518,6.973,148.278
C06212=1216.204,295.485,-67.003,-176.520,6.971,148.279
C06213=1216.208,295.236,-66.973,-176.523,6.968,148.279
C06214=1216.213,294.988,-66.944,-176.525,6.966,148.279
C06215=1216.217,294.740,-66.915,-176.527,6.963,148.279
C06216=1216.222,294.492,-66.886,-176.530,6.961,148.279
C06217=1216.226,294.243,-66.857,-176.533,6.958,148.279
C06218=1216.229,293.995,-66.828,-176.535,6.956,148.279
C06219=1216.235,293.747,-66.799,-176.537,6.954,148.279
C06220=1216.239,293.499,-66.770,-176.540,6.951,148.279
C06221=1216.243,293.251,-66.740,-176.542,6.949,148.279
C06222=1216.247,293.002,-66.711,-176.545,6.946,148.279
C06223=1216.252,292.753,-66.682,-176.547,6.943,148.279
C06224=1216.256,292.506,-66.653,-176.549,6.941,148.279
C06225=1216.261,292.257,-66.624,-176.552,6.938,148.279
C06226=1216.264,292.009,-66.596,-176.554,6.936,148.280
C06227=1216.268,291.761,-66.566,-176.557,6.933,148.280
C06228=1216.274,291.513,-66.538,-176.559,6.931,148.280
C06229=1216.278,291.264,-66.508,-176.561,6.929,148.280
C06230=1216.282,291.016,-66.479,-176.564,6.926,148.280
C06231=1216.286,290.767,-66.450,-176.567,6.924,148.280
C06232=1216.290,290.520,-66.422,-176.569,6.922,148.280
C06233=1216.295,290.271,-66.393,-176.571,6.919,148.280
C06234=1216.299,290.023,-66.363,-176.573,6.917,148.280
C06235=1216.304,289.775,-66.335,-176.577,6.914,148.281
C06236=1216.309,289.501,-66.303,-176.579,6.912,148.281
C06237=1216.314,289.227,-66.271,-176.581,6.909,148.281
C06238=1216.318,288.952,-66.239,-176.585,6.906,148.281
C06239=1216.323,288.678,-66.208,-176.587,6.903,148.281
C06240=1216.327,288.430,-66.178,-176.589,6.901,148.281
C06241=1216.331,288.181,-66.150,-176.592,6.899,148.281
C06242=1216.336,287.933,-66.121,-176.595,6.896,148.281
C06243=1216.340,287.684,-66.092,-176.597,6.893,148.281
C06244=1216.344,287.436,-66.064,-176.599,6.891,148.281
C06245=1216.349,287.188,-66.035,-176.602,6.889,148.282
C06246=1216.353,286.939,-66.006,-176.604,6.886,148.282
C06247=1216.358,286.691,-65.977,-176.607,6.883,148.282
C06248=1216.362,286.443,-65.949,-176.609,6.881,148.282
C06249=1216.366,286.194,-65.920,-176.612,6.879,148.282
C06250=1216.371,285.946,-65.891,-176.614,6.876,148.282
C06251=1216.375,285.698,-65.863,-176.616,6.874,148.282
C06252=1216.379,285.449,-65.834,-176.619,6.872,148.283
C06253=1216.383,285.201,-65.806,-176.622,6.869,148.283
C06254=1216.388,284.953,-65.777,-176.624,6.867,148.283
C06255=1216.392,284.704,-65.748,-176.626,6.865,148.283
C06256=1216.396,284.457,-65.720,-176.629,6.862,148.283
C06257=1216.401,284.208,-65.691,-176.631,6.860,148.283
C06258=1216.405,283.959,-65.663,-176.634,6.857,148.283
C06259=1216.410,283.711,-65.635,-176.636,6.855,148.283
C06260=1216.414,283.463,-65.606,-176.639,6.853,148.283
C06261=1216.418,283.215,-65.578,-176.641,6.850,148.283
C06262=1216.423,282.966,-65.549,-176.644,6.848,148.284
C06263=1216.427,282.719,-65.521,-176.646,6.845,148.284
C06264=1216.432,282.470,-65.492,-176.649,6.842,148.284
C06265=1216.436,282.221,-65.464,-176.651,6.841,148.284
C06266=1216.440,281.974,-65.435,-176.653,6.838,148.284
C06267=1216.445,281.725,-65.406,-176.656,6.835,148.284
C06268=1216.449,281.477,-65.379,-176.659,6.833,148.284
C06269=1216.453,281.228,-65.350,-176.661,6.831,148.285
C06270=1216.458,280.980,-65.322,-176.663,6.828,148.285
C06271=1216.462,280.731,-65.293,-176.666,6.826,148.285
C06272=1216.466,280.483,-65.265,-176.668,6.824,148.285
C06273=1216.471,280.234,-65.237,-176.671,6.821,148.285
C06274=1216.475,279.986,-65.209,-176.673,6.819,148.285
C06275=1216.480,279.738,-65.180,-176.676,6.817,148.285
C06276=1216.483,279.490,-65.151,-176.679,6.814,148.286
C06277=1216.488,279.242,-65.124,-176.681,6.812,148.286
C06278=1216.492,278.993,-65.095,-176.683,6.810,148.286
C06279=1216.497,278.745,-65.067,-176.686,6.807,148.286
C06280=1216.501,278.496,-65.038,-176.688,6.805,148.286
C06281=1216.505,278.248,-65.011,-176.690,6.803,148.286
C06282=1216.510,277.999,-64.982,-176.694,6.800,148.286
C06283=1216.515,277.751,-64.955,-176.696,6.798,148.286
C06284=1216.518,277.502,-64.927,-176.698,6.796,148.287
C06285=1216.523,277.254,-64.898,-176.701,6.793,148.287
C06286=1216.527,277.006,-64.870,-176.703,6.791,148.287
C06287=1216.532,276.758,-64.842,-176.706,6.789,148.287
C06288=1216.536,276.509,-64.814,-176.708,6.787,148.287
C06289=1216.540,276.261,-64.786,-176.711,6.784,148.287
C06290=1216.545,276.012,-64.757,-176.713,6.782,148.287
C06291=1216.549,275.764,-64.729,-176.715,6.780,148.288
C06292=1216.554,275.516,-64.702,-176.718,6.777,148.288
C06293=1216.558,275.267,-64.674,-176.721,6.775,148.288
C06294=1216.563,275.019,-64.646,-176.723,6.773,148.288
C06295=1216.566,274.770,-64.618,-176.726,6.770,148.288
C06296=1216.571,274.522,-64.590,-176.728,6.768,148.288
C06297=1216.575,274.274,-64.561,-176.731,6.766,148.289
C06298=1216.580,274.025,-64.534,-176.733,6.763,148.289
C06299=1216.584,273.777,-64.506,-176.736,6.761,148.289
C06300=1216.589,273.528,-64.477,-176.738,6.759,148.289
C06301=1216.593,273.280,-64.450,-176.741,6.757,148.289
C06302=1216.597,273.031,-64.422,-176.743,6.754,148.289
C06303=1216.602,272.783,-64.395,-176.746,6.752,148.290
C06304=1216.607,272.535,-64.366,-176.748,6.750,148.290
C06305=1216.610,272.287,-64.338,-176.750,6.747,148.290
C06306=1216.615,272.038,-64.311,-176.753,6.745,148.290
C06307=1216.619,271.789,-64.283,-176.755,6.742,148.290
C06308=1216.624,271.541,-64.254,-176.758,6.741,148.290
C06309=1216.629,271.293,-64.227,-176.761,6.737,148.290
C06310=1216.632,271.044,-64.199,-176.763,6.736,148.291
C06311=1216.637,270.796,-64.171,-176.765,6.733,148.291
C06312=1216.641,270.548,-64.144,-176.768,6.732,148.291
C06313=1216.646,270.299,-64.116,-176.771,6.729,148.291
C06314=1216.650,270.050,-64.089,-176.773,6.727,148.291
C06315=1216.655,269.803,-64.061,-176.775,6.724,148.291
C06316=1216.659,269.554,-64.033,-176.778,6.723,148.292
C06317=1216.663,269.306,-64.006,-176.781,6.720,148.292
C06318=1216.668,269.058,-63.978,-176.783,6.718,148.292
C06319=1216.672,268.808,-63.950,-176.786,6.715,148.292
C06320=1216.677,268.560,-63.922,-176.788,6.714,148.292
C06321=1216.681,268.312,-63.895,-176.791,6.711,148.292
C06322=1216.685,268.063,-63.867,-176.793,6.708,148.293
C06323=1216.690,267.815,-63.840,-176.796,6.706,148.293
C06324=1216.694,267.567,-63.812,-176.798,6.704,148.293
C06325=1216.698,267.318,-63.785,-176.801,6.702,148.293
C06326=1216.703,267.070,-63.757,-176.803,6.699,148.293
C06327=1216.707,266.821,-63.730,-176.806,6.697,148.294
C06328=1216.712,266.573,-63.703,-176.808,6.695,148.294
C06329=1216.716,266.324,-63.675,-176.811,6.693,148.294
C06330=1216.720,266.076,-63.647,-176.813,6.691,148.294
C06331=1216.725,265.828,-63.620,-176.816,6.689,148.294
C06332=1216.729,265.579,-63.593,-176.818,6.687,148.295
C06333=1216.734,265.330,-63.565,-176.821,6.684,148.295
C06334=1216.738,265.082,-63.537,-176.824,6.682,148.295
C06335=1216.743,264.833,-63.510,-176.826,6.680,148.295
C06336=1216.747,264.586,-63.482,-176.828,6.678,148.295
C06337=1216.751,264.336,-63.455,-176.831,6.675,148.295
C06338=1216.756,264.088,-63.427,-176.834,6.673,148.296
C06339=1216.761,263.839,-63.400,-176.836,6.671,148.296
C06340=1216.765,263.567,-63.371,-176.839,6.668,148.296
C06341=1216.770,263.294,-63.340,-176.841,6.666,148.296
C06342=1216.774,263.021,-63.310,-176.844,6.663,148.296
C06343=1216.780,262.749,-63.280,-176.847,6.661,148.297
C06344=1216.784,262.501,-63.254,-176.849,6.659,148.297
C06345=1216.788,262.252,-63.226,-176.852,6.656,148.297
C06346=1216.792,262.004,-63.198,-176.855,6.654,148.297
C06347=1216.797,261.755,-63.171,-176.857,6.652,148.297
C06348=1216.801,261.507,-63.144,-176.859,6.650,148.298
C06349=1216.806,261.258,-63.117,-176.862,6.647,148.298
C06350=1216.811,261.010,-63.090,-176.865,6.645,148.298
C06351=1216.815,260.762,-63.062,-176.867,6.643,148.298
C06352=1216.819,260.512,-63.035,-176.869,6.641,148.298
C06353=1216.824,260.264,-63.008,-176.872,6.639,148.299
C06354=1216.828,260.016,-62.981,-176.875,6.636,148.299
C06355=1216.832,259.767,-62.954,-176.877,6.634,148.299
C06356=1216.837,259.519,-62.927,-176.879,6.632,148.299
C06357=1216.842,259.270,-62.900,-176.882,6.630,148.299
C06358=1216.846,259.021,-62.873,-176.884,6.628,148.299
C06359=1216.850,258.773,-62.846,-176.887,6.626,148.300
C06360=1216.854,258.524,-62.819,-176.890,6.624,148.300
C06361=1216.859,258.277,-62.791,-176.892,6.621,148.300
C06362=1216.863,258.028,-62.764,-176.895,6.620,148.300
C06363=1216.868,257.780,-62.737,-176.897,6.617,148.301
C06364=1216.873,257.531,-62.710,-176.900,6.616,148.301
C06365=1216.877,257.283,-62.684,-176.903,6.613,148.301
C06366=1216.881,257.034,-62.657,-176.905,6.611,148.301
C06367=1216.885,256.785,-62.629,-176.907,6.609,148.301
C06368=1216.890,256.537,-62.602,-176.910,6.607,148.302
C06369=1216.894,256.289,-62.576,-176.912,6.605,148.302
C06370=1216.899,256.039,-62.549,-176.915,6.602,148.302
C06371=1216.903,255.791,-62.522,-176.917,6.600,148.302
C06372=1216.908,255.542,-62.495,-176.920,6.598,148.303
C06373=1216.912,255.294,-62.469,-176.922,6.596,148.303
C06374=1216.917,255.046,-62.442,-176.925,6.594,148.303
C06375=1216.921,254.797,-62.415,-176.927,6.592,148.303
C06376=1216.926,254.549,-62.388,-176.930,6.589,148.303
C06377=1216.930,254.301,-62.361,-176.933,6.587,148.304
C06378=1216.935,254.052,-62.334,-176.935,6.585,148.304
C06379=1216.940,253.803,-62.308,-176.938,6.583,148.304
C06380=1216.943,253.554,-62.281,-176.940,6.581,148.304
C06381=1216.947,253.306,-62.254,-176.942,6.579,148.304
C06382=1216.952,253.057,-62.227,-176.945,6.576,148.305
C06383=1216.956,252.809,-62.200,-176.948,6.574,148.305
C06384=1216.961,252.560,-62.173,-176.950,6.572,148.305
C06385=1216.965,252.312,-62.148,-176.953,6.570,148.305
C06386=1216.970,252.063,-62.120,-176.955,6.568,148.306
C06387=1216.974,251.815,-62.093,-176.958,6.566,148.306
C06388=1216.978,251.566,-62.067,-176.960,6.564,148.306
C06389=1216.983,251.317,-62.041,-176.963,6.562,148.306
C06390=1216.987,251.069,-62.014,-176.965,6.560,148.306
C06391=1216.992,250.821,-61.987,-176.968,6.558,148.307
C06392=1216.997,250.571,-61.961,-176.971,6.556,148.307
C06393=1217.001,250.323,-61.934,-176.973,6.554,148.307
C06394=1217.005,250.075,-61.907,-176.975,6.552,148.307
C06395=1217.009,249.826,-61.881,-176.978,6.550,148.308
C06396=1217.014,249.578,-61.854,-176.981,6.547,148.308
C06397=1217.018,249.329,-61.828,-176.983,6.545,148.308
C06398=1217.024,249.081,-61.802,-176.986,6.543,148.308
C06399=1217.028,248.832,-61.775,-176.988,6.541,148.308
C06400=1217.032,248.584,-61.748,-176.991,6.539,148.309
C06401=1217.037,248.335,-61.722,-176.993,6.537,148.309
C06402=1217.041,248.087,-61.696,-176.996,6.535,148.309
C06403=1217.046,247.838,-61.669,-176.998,6.533,148.310
C06404=1217.050,247.590,-61.643,-177.001,6.530,148.310
C06405=1217.055,247.341,-61.616,-177.003,6.528,148.310
C06406=1217.059,247.092,-61.590,-177.006,6.526,148.310
C06407=1217.063,246.844,-61.564,-177.009,6.524,148.310
C06408=1217.068,246.595,-61.537,-177.011,6.522,148.311
C06409=1217.072,246.347,-61.511,-177.013,6.520,148.311
C06410=1217.077,246.098,-61.484,-177.016,6.519,148.311
C06411=1217.081,245.850,-61.458,-177.018,6.516,148.311
C06412=1217.086,245.601,-61.432,-177.021,6.515,148.312
C06413=1217.090,245.352,-61.406,-177.024,6.512,148.312
C06414=1217.094,245.104,-61.380,-177.026,6.510,148.312
C06415=1217.099,244.855,-61.353,-177.029,6.508,148.312
C06416=1217.103,244.607,-61.327,-177.031,6.506,148.313
C06417=1217.108,244.358,-61.301,-177.034,6.504,148.313
C06418=1217.112,244.110,-61.274,-177.036,6.502,148.313
C06419=1217.116,243.861,-61.248,-177.039,6.500,148.313
C06420=1217.122,243.612,-61.222,-177.041,6.498,148.314
C06421=1217.126,243.364,-61.196,-177.044,6.496,148.314
C06422=1217.131,243.115,-61.170,-177.046,6.494,148.314
C06423=1217.135,242.866,-61.144,-177.049,6.491,148.314
C06424=1217.139,242.618,-61.117,-177.052,6.489,148.315
C06425=1217.144,242.369,-61.091,-177.054,6.487,148.315
C06426=1217.148,242.120,-61.065,-177.057,6.485,148.315
C06427=1217.153,241.873,-61.039,-177.059,6.484,148.315
C06428=1217.157,241.624,-61.013,-177.062,6.482,148.316
C06429=1217.162,241.375,-60.987,-177.064,6.480,148.316
C06430=1217.166,241.127,-60.961,-177.067,6.478,148.316
C06431=1217.170,240.878,-60.935,-177.069,6.476,148.316
C06432=1217.175,240.629,-60.909,-177.071,6.474,148.316
C06433=1217.180,240.381,-60.883,-177.074,6.472,148.317
C06434=1217.184,240.132,-60.857,-177.077,6.470,148.317
C06435=1217.188,239.884,-60.831,-177.080,6.467,148.317
C06436=1217.193,239.634,-60.805,-177.082,6.465,148.317
C06437=1217.198,239.386,-60.779,-177.085,6.463,148.318
C06438=1217.202,239.137,-60.753,-177.087,6.461,148.318
C06439=1217.206,238.889,-60.728,-177.090,6.459,148.318
C06440=1217.211,238.640,-60.701,-177.092,6.457,148.319
C06441=1217.216,238.392,-60.675,-177.095,6.455,148.319
C06442=1217.220,238.143,-60.649,-177.097,6.454,148.319
C06443=1217.224,237.894,-60.624,-177.100,6.452,148.319
C06444=1217.229,237.623,-60.596,-177.103,6.450,148.320
C06445=1217.234,237.352,-60.567,-177.106,6.447,148.320
C06446=1217.239,237.080,-60.539,-177.108,6.445,148.320
C06447=1217.244,236.809,-60.511,-177.110,6.443,148.320
C06448=1217.248,236.560,-60.484,-177.114,6.440,148.321
C06449=1217.252,236.312,-60.459,-177.116,6.438,148.321
C06450=1217.257,236.063,-60.433,-177.119,6.437,148.321
C06451=1217.262,235.815,-60.408,-177.122,6.435,148.322
C06452=1217.266,235.566,-60.382,-177.124,6.433,148.322
C06453=1217.271,235.317,-60.355,-177.126,6.431,148.322
C06454=1217.276,235.069,-60.330,-177.129,6.429,148.322
C06455=1217.280,234.820,-60.304,-177.132,6.427,148.323
C06456=1217.284,234.571,-60.279,-177.134,6.425,148.323
C06457=1217.288,234.322,-60.253,-177.136,6.423,148.323
C06458=1217.293,234.074,-60.227,-177.139,6.421,148.324
C06459=1217.297,233.825,-60.202,-177.142,6.419,148.324
C06460=1217.302,233.576,-60.177,-177.144,6.417,148.324
C06461=1217.307,233.328,-60.151,-177.146,6.415,148.324
C06462=1217.311,233.079,-60.126,-177.149,6.413,148.325
C06463=1217.315,232.830,-60.100,-177.152,6.411,148.325
C06464=1217.320,232.582,-60.074,-177.154,6.410,148.325
C06465=1217.324,232.333,-60.049,-177.157,6.408,148.326
C06466=1217.328,232.084,-60.023,-177.159,6.406,148.326
C06467=1217.333,231.836,-59.998,-177.162,6.404,148.326
C06468=1217.337,231.588,-59.972,-177.164,6.402,148.326
C06469=1217.343,231.339,-59.947,-177.167,6.400,148.327
C06470=1217.347,231.090,-59.921,-177.169,6.398,148.327
C06471=1217.351,230.841,-59.896,-177.172,6.396,148.327
C06472=1217.356,230.593,-59.870,-177.174,6.394,148.327
C06473=1217.360,230.344,-59.844,-177.177,6.392,148.328
C06474=1217.365,230.095,-59.819,-177.180,6.390,148.328
C06475=1217.369,229.847,-59.794,-177.183,6.388,148.328
C06476=1217.374,229.598,-59.768,-177.185,6.386,148.329
C06477=1217.378,229.350,-59.743,-177.188,6.384,148.329
C06478=1217.383,229.100,-59.718,-177.190,6.382,148.329
C06479=1217.387,228.852,-59.692,-177.193,6.380,148.329
C06480=1217.392,228.604,-59.667,-177.195,6.378,148.330
C06481=1217.397,228.354,-59.642,-177.198,6.376,148.330
C06482=1217.401,228.106,-59.616,-177.201,6.374,148.330
C06483=1217.406,227.857,-59.591,-177.203,6.373,148.331
C06484=1217.411,227.609,-59.566,-177.205,6.370,148.331
C06485=1217.415,227.360,-59.540,-177.208,6.368,148.331
C06486=1217.418,227.111,-59.515,-177.211,6.367,148.331
C06487=1217.424,226.863,-59.490,-177.213,6.365,148.332
C06488=1217.428,226.614,-59.465,-177.216,6.363,148.332
C06489=1217.433,226.366,-59.439,-177.219,6.361,148.332
C06490=1217.437,226.116,-59.414,-177.221,6.359,148.333
C06491=1217.442,225.868,-59.389,-177.223,6.357,148.333
C06492=1217.447,225.619,-59.364,-177.226,6.355,148.333
C06493=1217.451,225.371,-59.339,-177.229,6.353,148.333
C06494=1217.455,225.122,-59.313,-177.231,6.351,148.334
C06495=1217.460,224.873,-59.289,-177.234,6.350,148.334
C06496=1217.464,224.625,-59.263,-177.236,6.348,148.334
C06497=1217.469,224.376,-59.238,-177.239,6.346,148.335
C06498=1217.473,224.127,-59.213,-177.241,6.344,148.335
C06499=1217.478,223.879,-59.188,-177.244,6.342,148.335
C06500=1217.482,223.630,-59.163,-177.246,6.340,148.336
C06501=1217.487,223.381,-59.138,-177.249,6.338,148.336
C06502=1217.492,223.132,-59.112,-177.252,6.336,148.336
C06503=1217.496,222.884,-59.088,-177.254,6.334,148.336
C06504=1217.500,222.634,-59.063,-177.257,6.333,148.337
C06505=1217.505,222.386,-59.038,-177.260,6.331,148.337
C06506=1217.510,222.137,-59.013,-177.262,6.329,148.337
C06507=1217.514,221.889,-58.988,-177.264,6.327,148.338
C06508=1217.518,221.640,-58.963,-177.267,6.326,148.338
C06509=1217.523,221.392,-58.937,-177.269,6.324,148.338
C06510=1217.527,221.142,-58.913,-177.272,6.322,148.339
C06511=1217.532,220.894,-58.888,-177.274,6.320,148.339
C06512=1217.536,220.645,-58.862,-177.277,6.318,148.339
C06513=1217.541,220.397,-58.838,-177.280,6.316,148.340
C06514=1217.546,220.148,-58.814,-177.282,6.315,148.340
C06515=1217.550,219.899,-58.788,-177.285,6.313,148.340
C06516=1217.555,219.651,-58.764,-177.288,6.311,148.341
C06517=1217.559,219.401,-58.739,-177.290,6.309,148.341
C06518=1217.564,219.153,-58.714,-177.292,6.307,148.341
C06519=1217.568,218.904,-58.689,-177.295,6.305,148.341
C06520=1217.573,218.655,-58.664,-177.298,6.303,148.342
C06521=1217.578,218.406,-58.640,-177.300,6.301,148.342
C06522=1217.581,218.158,-58.615,-177.303,6.299,148.342
C06523=1217.587,217.909,-58.590,-177.306,6.298,148.343
C06524=1217.590,217.660,-58.565,-177.308,6.296,148.343
C06525=1217.596,217.411,-58.541,-177.311,6.294,148.343
C06526=1217.600,217.163,-58.515,-177.313,6.292,148.344
C06527=1217.604,216.914,-58.491,-177.316,6.290,148.344
C06528=1217.609,216.665,-58.466,-177.319,6.288,148.344
C06529=1217.614,216.417,-58.442,-177.321,6.286,148.345
C06530=1217.618,216.168,-58.417,-177.324,6.285,148.345
C06531=1217.623,215.919,-58.393,-177.327,6.283,148.345
C06532=1217.627,215.670,-58.367,-177.329,6.281,148.345
C06533=1217.632,215.422,-58.343,-177.331,6.279,148.346
C06534=1217.636,215.173,-58.319,-177.334,6.277,148.346
C06535=1217.641,214.924,-58.294,-177.337,6.275,148.346
C06536=1217.645,214.675,-58.270,-177.339,6.273,148.347
C06537=1217.650,214.427,-58.245,-177.342,6.271,148.347
C06538=1217.654,214.178,-58.220,-177.344,6.270,148.347
C06539=1217.659,213.929,-58.196,-177.347,6.269,148.348
C06540=1217.664,213.680,-58.172,-177.349,6.267,148.348
C06541=1217.668,213.431,-58.147,-177.352,6.265,148.348
C06542=1217.673,213.183,-58.123,-177.355,6.263,148.349
C06543=1217.677,212.934,-58.098,-177.357,6.261,148.349
C06544=1217.682,212.686,-58.074,-177.360,6.259,148.349
C06545=1217.686,212.436,-58.049,-177.362,6.257,148.350
C06546=1217.691,212.188,-58.025,-177.365,6.256,148.350
C06547=1217.695,211.939,-58.001,-177.368,6.254,148.350
C06548=1217.700,211.668,-57.974,-177.370,6.252,148.351
C06549=1217.705,211.398,-57.947,-177.373,6.250,148.351
C06550=1217.710,211.128,-57.920,-177.376,6.248,148.351
C06551=1217.715,210.858,-57.895,-177.379,6.246,148.352
C06552=1217.720,210.609,-57.870,-177.381,6.244,148.352
C06553=1217.724,210.360,-57.846,-177.384,6.243,148.352
C06554=1217.729,210.111,-57.821,-177.386,6.241,148.353
C06555=1217.734,209.863,-57.797,-177.389,6.239,148.353
C06556=1217.738,209.614,-57.773,-177.391,6.237,148.353
C06557=1217.742,209.365,-57.748,-177.394,6.235,148.354
C06558=1217.747,209.116,-57.724,-177.397,6.233,148.354
C06559=1217.752,208.867,-57.700,-177.399,6.232,148.354
C06560=1217.757,208.619,-57.676,-177.402,6.230,148.355
C06561=1217.760,208.369,-57.651,-177.405,6.228,148.355
C06562=1217.765,208.121,-57.627,-177.407,6.226,148.355
C06563=1217.770,207.872,-57.602,-177.410,6.224,148.356
C06564=1217.775,207.623,-57.579,-177.413,6.222,148.356
C06565=1217.779,207.375,-57.555,-177.415,6.221,148.357
C06566=1217.784,207.125,-57.530,-177.417,6.220,148.357
C06567=1217.788,206.877,-57.506,-177.420,6.218,148.357
C06568=1217.793,206.628,-57.483,-177.423,6.216,148.358
C06569=1217.798,206.379,-57.458,-177.425,6.214,148.358
C06570=1217.802,206.131,-57.434,-177.428,6.212,148.358
C06571=1217.807,205.882,-57.410,-177.430,6.210,148.359
C06572=1217.811,205.633,-57.386,-177.433,6.208,148.359
C06573=1217.816,205.384,-57.361,-177.436,6.207,148.359
C06574=1217.820,205.136,-57.337,-177.438,6.206,148.360
C06575=1217.825,204.887,-57.314,-177.440,6.204,148.360
C06576=1217.829,204.638,-57.290,-177.443,6.202,148.360
C06577=1217.834,204.390,-57.266,-177.446,6.200,148.361
C06578=1217.839,204.140,-57.241,-177.448,6.198,148.361
C06579=1217.843,203.891,-57.217,-177.451,6.196,148.361
C06580=1217.847,203.643,-57.193,-177.454,6.195,148.362
C06581=1217.852,203.394,-57.170,-177.456,6.193,148.362
C06582=1217.856,203.145,-57.146,-177.459,6.191,148.363
C06583=1217.862,202.896,-57.122,-177.462,6.190,148.363
C06584=1217.866,202.648,-57.098,-177.464,6.188,148.363
C06585=1217.870,202.398,-57.074,-177.467,6.186,148.364
C06586=1217.875,202.150,-57.050,-177.469,6.185,148.364
C06587=1217.879,201.901,-57.026,-177.472,6.183,148.364
C06588=1217.884,201.652,-57.003,-177.475,6.181,148.365
C06589=1217.888,201.404,-56.979,-177.477,6.179,148.365
C06590=1217.894,201.154,-56.955,-177.479,6.178,148.365
C06591=1217.898,200.906,-56.930,-177.482,6.176,148.366
C06592=1217.903,200.657,-56.907,-177.485,6.174,148.366
C06593=1217.907,200.408,-56.883,-177.487,6.173,148.366
C06594=1217.912,200.159,-56.860,-177.490,6.171,148.367
C06595=1217.917,199.910,-56.836,-177.493,6.169,148.367
C06596=1217.920,199.661,-56.812,-177.495,6.167,148.367
C06597=1217.925,199.412,-56.789,-177.497,6.166,148.368
C06598=1217.929,199.164,-56.764,-177.500,6.164,148.368
C06599=1217.934,198.915,-56.741,-177.503,6.162,148.368
C06600=1217.939,198.666,-56.717,-177.505,6.161,148.369
C06601=1217.943,198.417,-56.694,-177.508,6.159,148.369
C06602=1217.948,198.168,-56.670,-177.511,6.157,148.369
C06603=1217.953,197.920,-56.646,-177.513,6.156,148.370
C06604=1217.958,197.671,-56.622,-177.515,6.154,148.370
C06605=1217.962,197.422,-56.599,-177.518,6.153,148.371
C06606=1217.967,197.173,-56.575,-177.521,6.151,148.371
C06607=1217.972,196.924,-56.552,-177.524,6.149,148.371
C06608=1217.976,196.675,-56.528,-177.526,6.147,148.372
C06609=1217.981,196.427,-56.504,-177.529,6.146,148.372
C06610=1217.985,196.178,-56.481,-177.531,6.144,148.373
C06611=1217.989,195.929,-56.458,-177.534,6.142,148.373
C06612=1217.994,195.681,-56.434,-177.536,6.140,148.373
C06613=1217.998,195.431,-56.411,-177.539,6.139,148.374
C06614=1218.003,195.182,-56.387,-177.542,6.137,148.374
C06615=1218.008,194.933,-56.364,-177.544,6.136,148.374
C06616=1218.012,194.685,-56.340,-177.546,6.134,148.375
C06617=1218.017,194.436,-56.316,-177.549,6.132,148.375
C06618=1218.022,194.187,-56.293,-177.552,6.131,148.376
C06619=1218.026,193.938,-56.270,-177.555,6.129,148.376
C06620=1218.031,193.689,-56.246,-177.557,6.128,148.376
C06621=1218.035,193.440,-56.222,-177.560,6.126,148.377
C06622=1218.040,193.191,-56.199,-177.562,6.124,148.377
C06623=1218.045,192.942,-56.175,-177.565,6.122,148.377
C06624=1218.050,192.693,-56.152,-177.568,6.120,148.378
C06625=1218.054,192.445,-56.130,-177.570,6.119,148.378
C06626=1218.059,192.196,-56.106,-177.572,6.118,148.378
C06627=1218.063,191.947,-56.083,-177.575,6.116,148.379
C06628=1218.068,191.698,-56.060,-177.578,6.114,148.379
C06629=1218.073,191.450,-56.036,-177.581,6.112,148.380
C06630=1218.077,191.201,-56.012,-177.583,6.111,148.380
C06631=1218.082,190.952,-55.989,-177.585,6.110,148.380
C06632=1218.086,190.703,-55.966,-177.588,6.108,148.381
C06633=1218.091,190.454,-55.943,-177.591,6.106,148.381
C06634=1218.095,190.205,-55.919,-177.593,6.104,148.381
C06635=1218.100,189.956,-55.896,-177.595,6.103,148.382
C06636=1218.105,189.708,-55.873,-177.598,6.101,148.382
C06637=1218.109,189.459,-55.850,-177.601,6.099,148.382
C06638=1218.114,189.210,-55.827,-177.604,6.098,148.383
C06639=1218.119,188.961,-55.804,-177.607,6.096,148.383
C06640=1218.123,188.712,-55.780,-177.609,6.095,148.384
C06641=1218.127,188.463,-55.757,-177.611,6.093,148.384
C06642=1218.132,188.214,-55.734,-177.614,6.091,148.384
C06643=1218.137,187.965,-55.711,-177.617,6.090,148.385
C06644=1218.142,187.717,-55.688,-177.619,6.089,148.385
C06645=1218.146,187.468,-55.665,-177.621,6.087,148.386
C06646=1218.151,187.219,-55.642,-177.624,6.085,148.386
C06647=1218.156,186.969,-55.619,-177.627,6.083,148.386
C06648=1218.160,186.720,-55.596,-177.630,6.082,148.387
C06649=1218.164,186.472,-55.573,-177.632,6.081,148.387
C06650=1218.170,186.223,-55.550,-177.635,6.079,148.388
C06651=1218.174,185.974,-55.526,-177.637,6.077,148.388
C06652=1218.179,185.705,-55.502,-177.640,6.075,148.388
C06653=1218.184,185.435,-55.477,-177.643,6.074,148.389
C06654=1218.190,185.165,-55.452,-177.646,6.072,148.389
C06655=1218.194,184.896,-55.428,-177.648,6.070,148.390
C06656=1218.199,184.647,-55.404,-177.651,6.069,148.390
C06657=1218.203,184.398,-55.381,-177.653,6.067,148.390
C06658=1218.208,184.149,-55.358,-177.656,6.066,148.391
C06659=1218.213,183.899,-55.335,-177.659,6.064,148.391
C06660=1218.217,183.651,-55.313,-177.661,6.063,148.392
C06661=1218.222,183.402,-55.290,-177.664,6.061,148.392
C06662=1218.227,183.153,-55.266,-177.666,6.059,148.392
C06663=1218.231,182.904,-55.244,-177.669,6.058,148.393
C06664=1218.236,182.656,-55.221,-177.671,6.057,148.393
C06665=1218.240,182.407,-55.198,-177.674,6.055,148.394
C06666=1218.245,182.158,-55.175,-177.677,6.053,148.394
C06667=1218.250,181.908,-55.152,-177.679,6.051,148.394
C06668=1218.254,181.660,-55.130,-177.681,6.050,148.395
C06669=1218.259,181.411,-55.107,-177.685,6.049,148.395
C06670=1218.263,181.162,-55.085,-177.687,6.047,148.396
C06671=1218.268,180.913,-55.061,-177.690,6.045,148.396
C06672=1218.273,180.665,-55.039,-177.692,6.044,148.396
C06673=1218.278,180.415,-55.016,-177.695,6.042,148.397
C06674=1218.282,180.166,-54.994,-177.697,6.040,148.397
C06675=1218.287,179.917,-54.971,-177.700,6.040,148.398
C06676=1218.291,179.669,-54.948,-177.703,6.038,148.398
C06677=1218.296,179.420,-54.925,-177.705,6.036,148.398
C06678=1218.300,179.170,-54.903,-177.708,6.034,148.399
C06679=1218.305,178.922,-54.880,-177.710,6.033,148.399
C06680=1218.310,178.673,-54.858,-177.713,6.031,148.399
C06681=1218.314,178.424,-54.835,-177.716,6.030,148.400
C06682=1218.319,178.175,-54.813,-177.718,6.029,148.400
C06683=1218.324,177.926,-54.790,-177.720,6.027,148.401
C06684=1218.328,177.677,-54.768,-177.723,6.025,148.401
C06685=1218.333,177.427,-54.744,-177.726,6.023,148.402
C06686=1218.338,177.179,-54.723,-177.728,6.023,148.402
C06687=1218.342,176.930,-54.700,-177.731,6.021,148.402
C06688=1218.347,176.680,-54.677,-177.734,6.019,148.403
C06689=1218.351,176.432,-54.655,-177.736,6.018,148.403
C06690=1218.356,176.183,-54.632,-177.738,6.016,148.404
C06691=1218.361,175.935,-54.610,-177.742,6.015,148.404
C06692=1218.366,175.685,-54.587,-177.744,6.014,148.405
C06693=1218.370,175.436,-54.564,-177.746,6.012,148.405
C06694=1218.375,175.188,-54.543,-177.749,6.010,148.405
C06695=1218.380,174.938,-54.520,-177.752,6.008,148.406
C06696=1218.384,174.689,-54.497,-177.754,6.008,148.406
C06697=1218.389,174.441,-54.476,-177.757,6.006,148.407
C06698=1218.393,174.192,-54.452,-177.760,6.004,148.407
C06699=1218.398,173.943,-54.430,-177.762,6.003,148.407
C06700=1218.403,173.693,-54.408,-177.764,6.001,148.408
C06701=1218.407,173.445,-54.385,-177.767,6.000,148.408
C06702=1218.412,173.196,-54.363,-177.770,5.999,148.409
C06703=1218.417,172.946,-54.341,-177.772,5.997,148.409
C06704=1218.421,172.698,-54.318,-177.775,5.995,148.409
C06705=1218.426,172.449,-54.296,-177.777,5.994,148.410
C06706=1218.430,172.200,-54.274,-177.780,5.993,148.410
C06707=1218.435,171.951,-54.251,-177.783,5.991,148.411
C06708=1218.440,171.702,-54.229,-177.785,5.990,148.411
C06709=1218.444,171.453,-54.208,-177.787,5.988,148.411
C06710=1218.449,171.204,-54.185,-177.791,5.986,148.412
C06711=1218.454,170.956,-54.162,-177.793,5.986,148.412
C06712=1218.458,170.706,-54.140,-177.795,5.984,148.413
C06713=1218.463,170.457,-54.118,-177.798,5.982,148.413
C06714=1218.468,170.208,-54.096,-177.801,5.981,148.414
C06715=1218.472,169.959,-54.074,-177.803,5.979,148.414
C06716=1218.477,169.711,-54.052,-177.806,5.978,148.414
C06717=1218.481,169.461,-54.030,-177.808,5.977,148.415
C06718=1218.487,169.212,-54.007,-177.811,5.975,148.415
C06719=1218.491,168.963,-53.985,-177.814,5.973,148.416
C06720=1218.496,168.714,-53.964,-177.816,5.972,148.416
C06721=1218.500,168.465,-53.942,-177.819,5.970,148.417
C06722=1218.505,168.216,-53.920,-177.821,5.970,148.417
C06723=1218.510,167.967,-53.897,-177.824,5.968,148.418
C06724=1218.515,167.719,-53.875,-177.827,5.966,148.418
C06725=1218.519,167.469,-53.853,-177.829,5.965,148.418
C06726=1218.524,167.221,-53.831,-177.832,5.964,148.419
C06727=1218.528,166.971,-53.809,-177.834,5.962,148.419
C06728=1218.533,166.723,-53.787,-177.837,5.961,148.420
C06729=1218.538,166.473,-53.765,-177.839,5.959,148.420
C06730=1218.543,166.225,-53.743,-177.842,5.958,148.421
C06731=1218.547,165.975,-53.721,-177.844,5.957,148.421
C06732=1218.552,165.727,-53.699,-177.847,5.955,148.421
C06733=1218.556,165.477,-53.677,-177.849,5.954,148.422
C06734=1218.561,165.229,-53.656,-177.852,5.952,148.422
C06735=1218.565,164.979,-53.634,-177.855,5.950,148.423
C06736=1218.570,164.731,-53.612,-177.857,5.949,148.423
C06737=1218.575,164.481,-53.590,-177.860,5.948,148.423
C06738=1218.580,164.232,-53.568,-177.863,5.946,148.424
C06739=1218.585,163.984,-53.546,-177.865,5.945,148.424
C06740=1218.589,163.734,-53.524,-177.868,5.943,148.425
C06741=1218.594,163.486,-53.502,-177.870,5.943,148.425
C06742=1218.598,163.236,-53.480,-177.873,5.941,148.426
C06743=1218.603,162.988,-53.458,-177.876,5.939,148.426
C06744=1218.608,162.738,-53.436,-177.878,5.938,148.427
C06745=1218.612,162.490,-53.415,-177.881,5.937,148.427
C06746=1218.617,162.241,-53.393,-177.883,5.936,148.428
C06747=1218.622,161.991,-53.372,-177.886,5.934,148.428
C06748=1218.627,161.742,-53.350,-177.888,5.932,148.428
C06749=1218.631,161.493,-53.328,-177.891,5.931,148.429
C06750=1218.636,161.245,-53.306,-177.894,5.930,148.429
C06751=1218.641,160.996,-53.285,-177.896,5.929,148.430
C06752=1218.645,160.747,-53.262,-177.899,5.927,148.430
C06753=1218.650,160.497,-53.242,-177.901,5.925,148.431
C06754=1218.654,160.248,-53.219,-177.904,5.924,148.431
C06755=1218.659,159.999,-53.198,-177.907,5.923,148.432
C06756=1218.665,159.730,-53.174,-177.909,5.921,148.432
C06757=1218.669,159.462,-53.151,-177.911,5.920,148.432
C06758=1218.675,159.192,-53.128,-177.915,5.919,148.433
C06759=1218.679,158.923,-53.105,-177.917,5.917,148.433
C06760=1218.684,158.674,-53.083,-177.920,5.915,148.434
C06761=1218.689,158.425,-53.061,-177.923,5.914,148.434
C06762=1218.693,158.176,-53.039,-177.925,5.912,148.435
C06763=1218.699,157.927,-53.018,-177.928,5.912,148.435
C06764=1218.703,157.678,-52.996,-177.930,5.910,148.436
C06765=1218.708,157.429,-52.975,-177.933,5.908,148.436
C06766=1218.713,157.180,-52.954,-177.936,5.908,148.437
C06767=1218.717,156.931,-52.932,-177.938,5.906,148.437
C06768=1218.721,156.682,-52.911,-177.940,5.905,148.437
C06769=1218.727,156.433,-52.890,-177.944,5.903,148.438
C06770=1218.731,156.184,-52.868,-177.946,5.902,148.438
C06771=1218.736,155.935,-52.846,-177.948,5.900,148.439
C06772=1218.741,155.686,-52.825,-177.952,5.899,148.439
C06773=1218.746,155.437,-52.803,-177.954,5.898,148.440
C06774=1218.750,155.187,-52.782,-177.956,5.896,148.440
C06775=1218.754,154.939,-52.761,-177.959,5.896,148.441
C06776=1218.759,154.690,-52.739,-177.962,5.894,148.441
C06777=1218.764,154.440,-52.718,-177.964,5.893,148.442
C06778=1218.769,154.192,-52.696,-177.967,5.891,148.442
C06779=1218.774,153.942,-52.675,-177.969,5.890,148.443
C06780=1218.778,153.694,-52.654,-177.972,5.889,148.443
C06781=1218.783,153.444,-52.633,-177.975,5.887,148.443
C06782=1218.788,153.195,-52.611,-177.977,5.886,148.444
C06783=1218.793,152.946,-52.590,-177.980,5.884,148.444
C06784=1218.798,152.698,-52.568,-177.982,5.884,148.445
C06785=1218.801,152.448,-52.548,-177.985,5.882,148.445
C06786=1218.806,152.199,-52.526,-177.987,5.881,148.446
C06787=1218.811,151.950,-52.505,-177.990,5.879,148.446
C06788=1218.816,151.701,-52.483,-177.992,5.878,148.447
C06789=1218.821,151.452,-52.463,-177.995,5.877,148.447
C06790=1218.825,151.203,-52.441,-177.997,5.876,148.448
C06791=1218.830,150.954,-52.420,-178.000,5.874,148.448
C06792=1218.835,150.705,-52.398,-178.002,5.873,148.448
C06793=1218.839,150.456,-52.378,-178.005,5.872,148.449
C06794=1218.844,150.206,-52.357,-178.008,5.870,148.449
C06795=1218.849,149.958,-52.335,-178.010,5.869,148.450
C06796=1218.853,149.709,-52.315,-178.013,5.867,148.450
C06797=1218.858,149.460,-52.293,-178.015,5.866,148.451
C06798=1218.863,149.211,-52.272,-178.018,5.865,148.451
C06799=1218.867,148.961,-52.251,-178.021,5.864,148.452
C06800=1218.872,148.712,-52.229,-178.023,5.862,148.452
C06801=1218.877,148.463,-52.208,-178.026,5.862,148.453
C06802=1218.882,148.214,-52.188,-178.029,5.860,148.453
C06803=1218.887,147.966,-52.166,-178.031,5.859,148.454
C06804=1218.892,147.716,-52.145,-178.034,5.857,148.454
C06805=1218.896,147.467,-52.125,-178.036,5.856,148.455
C06806=1218.901,147.217,-52.104,-178.039,5.854,148.455
C06807=1218.905,146.969,-52.083,-178.041,5.854,148.456
C06808=1218.910,146.720,-52.062,-178.044,5.852,148.456
C06809=1218.915,146.471,-52.041,-178.047,5.851,148.457
C06810=1218.919,146.222,-52.020,-178.049,5.850,148.457
C06811=1218.925,145.973,-51.999,-178.051,5.849,148.457
C06812=1218.929,145.724,-51.978,-178.054,5.847,148.458
C06813=1218.934,145.474,-51.957,-178.057,5.846,148.458
C06814=1218.939,145.225,-51.936,-178.059,5.844,148.459
C06815=1218.943,144.977,-51.915,-178.062,5.844,148.459
C06816=1218.948,144.727,-51.894,-178.064,5.842,148.460
C06817=1218.952,144.478,-51.874,-178.067,5.841,148.460
C06818=1218.958,144.229,-51.853,-178.070,5.839,148.461
C06819=1218.962,143.980,-51.832,-178.072,5.839,148.461
C06820=1218.967,143.731,-51.811,-178.075,5.837,148.462
C06821=1218.971,143.483,-51.790,-178.077,5.836,148.462
C06822=1218.976,143.233,-51.769,-178.080,5.835,148.463
C06823=1218.980,142.984,-51.749,-178.082,5.834,148.463
C06824=1218.986,142.734,-51.728,-178.085,5.832,148.463
C06825=1218.990,142.485,-51.707,-178.088,5.831,148.464
C06826=1218.995,142.236,-51.686,-178.090,5.829,148.464
C06827=1219.000,141.987,-51.666,-178.093,5.829,148.465
C06828=1219.005,141.738,-51.645,-178.096,5.827,148.466
C06829=1219.009,141.489,-51.624,-178.098,5.826,148.466
C06830=1219.014,141.240,-51.604,-178.101,5.825,148.467
C06831=1219.019,140.991,-51.583,-178.103,5.824,148.467
C06832=1219.024,140.742,-51.561,-178.106,5.822,148.468
C06833=1219.028,140.493,-51.541,-178.108,5.821,148.468
C06834=1219.033,140.244,-51.521,-178.111,5.819,148.468
C06835=1219.038,139.995,-51.500,-178.114,5.819,148.469
C06836=1219.042,139.746,-51.479,-178.116,5.818,148.469
C06837=1219.047,139.497,-51.458,-178.119,5.816,148.470
C06838=1219.052,139.248,-51.438,-178.121,5.815,148.470
C06839=1219.057,138.998,-51.418,-178.124,5.814,148.471
C06840=1219.062,138.749,-51.397,-178.126,5.813,148.471
C06841=1219.066,138.500,-51.377,-178.129,5.811,148.472
C06842=1219.071,138.251,-51.356,-178.131,5.810,148.472
C06843=1219.076,138.002,-51.336,-178.134,5.809,148.473
C06844=1219.080,137.753,-51.315,-178.137,5.808,148.473
C06845=1219.085,137.504,-51.294,-178.139,5.806,148.474
C06846=1219.090,137.255,-51.274,-178.142,5.806,148.474
C06847=1219.095,137.005,-51.253,-178.144,5.805,148.475
C06848=1219.099,136.756,-51.233,-178.147,5.803,148.475
C06849=1219.104,136.508,-51.212,-178.149,5.802,148.476
C06850=1219.109,136.258,-51.192,-178.152,5.800,148.476
C06851=1219.114,136.009,-51.172,-178.155,5.800,148.477
C06852=1219.118,135.760,-51.151,-178.157,5.798,148.477
C06853=1219.123,135.511,-51.131,-178.160,5.797,148.478
C06854=1219.128,135.262,-51.110,-178.163,5.796,148.478
C06855=1219.132,135.013,-51.090,-178.165,5.795,148.479
C06856=1219.137,134.763,-51.070,-178.167,5.794,148.479
C06857=1219.142,134.514,-51.049,-178.170,5.792,148.480
C06858=1219.147,134.265,-51.029,-178.173,5.791,148.480
C06859=1219.151,134.016,-51.008,-178.175,5.790,148.481
C06860=1219.157,133.747,-50.987,-178.178,5.789,148.481
C06861=1219.162,133.479,-50.964,-178.181,5.788,148.482
C06862=1219.167,133.210,-50.943,-178.184,5.786,148.482
C06863=1219.172,132.941,-50.920,-178.186,5.785,148.483
C06864=1219.177,132.692,-50.901,-178.189,5.783,148.483
C06865=1219.182,132.443,-50.881,-178.192,5.783,148.484
C06866=1219.187,132.194,-50.860,-178.194,5.782,148.484
C06867=1219.191,131.945,-50.839,-178.197,5.780,148.485
C06868=1219.196,131.695,-50.820,-178.199,5.779,148.485
C06869=1219.200,131.446,-50.799,-178.202,5.778,148.486
C06870=1219.205,131.197,-50.779,-178.204,5.777,148.486
C06871=1219.210,130.947,-50.759,-178.207,5.775,148.487
C06872=1219.215,130.699,-50.738,-178.210,5.775,148.487
C06873=1219.220,130.450,-50.718,-178.212,5.774,148.488
C06874=1219.224,130.201,-50.699,-178.215,5.772,148.488
C06875=1219.229,129.952,-50.678,-178.217,5.771,148.489
C06876=1219.234,129.702,-50.659,-178.220,5.770,148.489
C06877=1219.239,129.453,-50.638,-178.222,5.769,148.490
C06878=1219.243,129.204,-50.617,-178.225,5.768,148.490
C06879=1219.248,128.954,-50.598,-178.228,5.766,148.491
C06880=1219.253,128.706,-50.578,-178.230,5.766,148.491
C06881=1219.258,128.457,-50.558,-178.233,5.764,148.492
C06882=1219.262,128.208,-50.538,-178.235,5.763,148.493
C06883=1219.267,127.958,-50.518,-178.238,5.762,148.493
C06884=1219.271,127.709,-50.498,-178.241,5.761,148.494
C06885=1219.276,127.460,-50.478,-178.243,5.760,148.494
C06886=1219.282,127.211,-50.457,-178.246,5.758,148.495
C06887=1219.287,126.961,-50.438,-178.248,5.757,148.495
C06888=1219.291,126.712,-50.417,-178.251,5.757,148.496
C06889=1219.296,126.463,-50.398,-178.253,5.755,148.496
C06890=1219.300,126.214,-50.377,-178.256,5.754,148.497
C06891=1219.306,125.965,-50.358,-178.259,5.753,148.497
C06892=1219.310,125.716,-50.338,-178.261,5.752,148.498
C06893=1219.315,125.467,-50.318,-178.263,5.751,148.498
C06894=1219.319,125.218,-50.298,-178.267,5.750,148.499
C06895=1219.324,124.968,-50.278,-178.269,5.749,148.499
C06896=1219.329,124.720,-50.258,-178.271,5.748,148.500
C06897=1219.334,124.470,-50.238,-178.274,5.746,148.500
C06898=1219.339,124.221,-50.219,-178.277,5.746,148.501
C06899=1219.343,123.972,-50.198,-178.279,5.744,148.501
C06900=1219.348,123.723,-50.179,-178.282,5.743,148.502
C06901=1219.353,123.473,-50.159,-178.284,5.742,148.502
C06902=1219.357,123.224,-50.139,-178.287,5.741,148.503
C06903=1219.362,122.975,-50.119,-178.289,5.740,148.503
C06904=1219.368,122.726,-50.100,-178.292,5.739,148.504
C06905=1219.372,122.477,-50.080,-178.295,5.737,148.504
C06906=1219.377,122.227,-50.060,-178.297,5.737,148.505
C06907=1219.381,121.978,-50.040,-178.299,5.736,148.505
C06908=1219.387,121.730,-50.020,-178.303,5.734,148.506
C06909=1219.391,121.480,-50.001,-178.305,5.733,148.506
C06910=1219.396,121.230,-49.981,-178.308,5.732,148.507
C06911=1219.401,120.982,-49.961,-178.310,5.731,148.507
C06912=1219.406,120.733,-49.941,-178.313,5.730,148.508
C06913=1219.411,120.483,-49.922,-178.315,5.729,148.508
C06914=1219.415,120.234,-49.903,-178.318,5.728,148.509
C06915=1219.420,119.986,-49.883,-178.320,5.727,148.510
C06916=1219.424,119.736,-49.863,-178.323,5.726,148.510
C06917=1219.429,119.486,-49.843,-178.326,5.725,148.511
C06918=1219.434,119.238,-49.824,-178.328,5.724,148.511
C06919=1219.439,118.988,-49.804,-178.331,5.723,148.512
C06920=1219.444,118.739,-49.784,-178.333,5.722,148.512
C06921=1219.449,118.490,-49.765,-178.336,5.721,148.513
C06922=1219.454,118.241,-49.745,-178.338,5.719,148.513
C06923=1219.458,117.991,-49.726,-178.341,5.719,148.514
C06924=1219.463,117.742,-49.707,-178.343,5.718,148.514
C06925=1219.468,117.493,-49.687,-178.346,5.716,148.515
C06926=1219.472,117.244,-49.667,-178.348,5.715,148.515
C06927=1219.478,116.995,-49.647,-178.351,5.715,148.516
C06928=1219.482,116.746,-49.628,-178.354,5.713,148.516
C06929=1219.486,116.496,-49.609,-178.356,5.712,148.517
C06930=1219.492,116.247,-49.589,-178.359,5.712,148.518
C06931=1219.496,115.998,-49.570,-178.362,5.710,148.518
C06932=1219.502,115.749,-49.550,-178.364,5.709,148.519
C06933=1219.506,115.499,-49.531,-178.366,5.708,148.519
C06934=1219.510,115.250,-49.512,-178.370,5.707,148.520
C06935=1219.516,115.001,-49.492,-178.372,5.706,148.520
C06936=1219.521,114.752,-49.473,-178.374,5.705,148.521
C06937=1219.525,114.502,-49.453,-178.377,5.703,148.521
C06938=1219.530,114.254,-49.434,-178.380,5.703,148.522
C06939=1219.535,114.004,-49.415,-178.382,5.702,148.522
C06940=1219.540,113.755,-49.395,-178.385,5.700,148.523
C06941=1219.545,113.506,-49.376,-178.388,5.700,148.523
C06942=1219.549,113.256,-49.357,-178.390,5.699,148.524
C06943=1219.554,113.007,-49.337,-178.392,5.698,148.524
C06944=1219.559,112.758,-49.318,-178.395,5.696,148.525
C06945=1219.564,112.509,-49.298,-178.398,5.696,148.525
C06946=1219.568,112.260,-49.279,-178.400,5.695,148.526
C06947=1219.574,112.011,-49.260,-178.403,5.693,148.527
C06948=1219.578,111.761,-49.240,-178.405,5.693,148.527
C06949=1219.582,111.512,-49.221,-178.408,5.692,148.528
C06950=1219.588,111.263,-49.202,-178.411,5.690,148.528
C06951=1219.592,111.014,-49.182,-178.413,5.690,148.529
C06952=1219.597,110.765,-49.164,-178.415,5.689,148.529
C06953=1219.602,110.516,-49.144,-178.418,5.688,148.530
C06954=1219.607,110.266,-49.125,-178.421,5.687,148.530
C06955=1219.611,110.017,-49.106,-178.423,5.686,148.531
C06956=1219.617,109.768,-49.087,-178.426,5.685,148.531
C06957=1219.621,109.518,-49.067,-178.429,5.684,148.532
C06958=1219.626,109.270,-49.049,-178.431,5.683,148.532
C06959=1219.631,109.020,-49.029,-178.433,5.682,148.533
C06960=1219.635,108.772,-49.010,-178.436,5.681,148.534
C06961=1219.640,108.521,-48.991,-178.439,5.680,148.534
C06962=1219.646,108.273,-48.972,-178.441,5.679,148.535
C06963=1219.650,108.023,-48.953,-178.443,5.678,148.535
C06964=1219.655,107.755,-48.932,-178.447,5.677,148.536
C06965=1219.661,107.486,-48.912,-178.449,5.676,148.536
C06966=1219.666,107.218,-48.891,-178.452,5.675,148.537
C06967=1219.671,106.949,-48.872,-178.455,5.674,148.538
C06968=1219.676,106.700,-48.852,-178.457,5.673,148.538
C06969=1219.681,106.451,-48.833,-178.460,5.672,148.539
C06970=1219.685,106.202,-48.814,-178.463,5.671,148.539
C06971=1219.690,105.952,-48.795,-178.465,5.670,148.540
C06972=1219.695,105.703,-48.776,-178.468,5.669,148.540
C06973=1219.700,105.454,-48.757,-178.470,5.668,148.541
C06974=1219.705,105.205,-48.739,-178.473,5.667,148.541
C06975=1219.709,104.955,-48.719,-178.475,5.666,148.542
C06976=1219.714,104.707,-48.700,-178.478,5.665,148.543
C06977=1219.720,104.457,-48.682,-178.481,5.664,148.543
C06978=1219.724,104.208,-48.663,-178.483,5.663,148.544
C06979=1219.729,103.959,-48.643,-178.486,5.662,148.544
C06980=1219.733,103.709,-48.625,-178.488,5.661,148.545
C06981=1219.739,103.460,-48.606,-178.491,5.660,148.545
C06982=1219.743,103.211,-48.587,-178.494,5.659,148.546
C06983=1219.748,102.962,-48.568,-178.496,5.659,148.546
C06984=1219.753,102.713,-48.549,-178.499,5.657,148.547
C06985=1219.758,102.463,-48.530,-178.501,5.656,148.547
C06986=1219.762,102.214,-48.512,-178.504,5.656,148.548
C06987=1219.767,101.965,-48.492,-178.506,5.655,148.549
C06988=1219.772,101.715,-48.474,-178.509,5.653,148.549
C06989=1219.777,101.467,-48.455,-178.512,5.653,148.550
C06990=1219.782,101.217,-48.436,-178.514,5.652,148.550
C06991=1219.786,100.968,-48.418,-178.516,5.651,148.551
C06992=1219.791,100.718,-48.399,-178.519,5.650,148.551
C06993=1219.796,100.469,-48.380,-178.522,5.649,148.552
C06994=1219.801,100.220,-48.362,-178.524,5.648,148.553
C06995=1219.806,99.971,-48.342,-178.527,5.647,148.553
C06996=1219.811,99.722,-48.324,-178.529,5.646,148.554
C06997=1219.815,99.472,-48.305,-178.532,5.645,148.554
C06998=1219.820,99.223,-48.287,-178.535,5.644,148.555
C06999=1219.825,98.974,-48.268,-178.537,5.644,148.555
C07000=1219.830,98.724,-48.249,-178.540,5.643,148.556
C07001=1219.835,98.475,-48.231,-178.543,5.641,148.557
C07002=1219.839,98.226,-48.213,-178.545,5.641,148.557
C07003=1219.844,97.976,-48.194,-178.547,5.640,148.558
C07004=1219.849,97.728,-48.175,-178.550,5.639,148.558
C07005=1219.854,97.478,-48.157,-178.552,5.638,148.559
C07006=1219.859,97.229,-48.137,-178.555,5.637,148.559
C07007=1219.864,96.980,-48.119,-178.558,5.636,148.560
C07008=1219.869,96.730,-48.101,-178.560,5.635,148.560
C07009=1219.873,96.481,-48.082,-178.563,5.635,148.561
C07010=1219.878,96.232,-48.064,-178.565,5.633,148.561
C07011=1219.883,95.983,-48.046,-178.568,5.632,148.562
C07012=1219.888,95.734,-48.026,-178.571,5.632,148.563
C07013=1219.893,95.484,-48.008,-178.573,5.631,148.563
C07014=1219.898,95.235,-47.990,-178.575,5.630,148.564
C07015=1219.902,94.986,-47.971,-178.579,5.629,148.564
C07016=1219.907,94.736,-47.952,-178.581,5.628,148.565
C07017=1219.912,94.487,-47.934,-178.583,5.627,148.566
C07018=1219.917,94.238,-47.916,-178.586,5.627,148.566
C07019=1219.922,93.989,-47.898,-178.588,5.626,148.567
C07020=1219.927,93.739,-47.879,-178.591,5.624,148.567
C07021=1219.932,93.490,-47.861,-178.594,5.624,148.568
C07022=1219.936,93.241,-47.842,-178.596,5.623,148.568
C07023=1219.941,92.991,-47.824,-178.599,5.622,148.569
C07024=1219.946,92.742,-47.806,-178.601,5.622,148.570
C07025=1219.951,92.492,-47.787,-178.604,5.620,148.570
C07026=1219.956,92.243,-47.769,-178.607,5.619,148.571
C07027=1219.960,91.994,-47.750,-178.609,5.619,148.571
C07028=1219.965,91.745,-47.732,-178.611,5.618,148.572
C07029=1219.970,91.496,-47.714,-178.614,5.617,148.572
C07030=1219.976,91.246,-47.696,-178.617,5.616,148.573
C07031=1219.981,90.997,-47.678,-178.619,5.615,148.573
C07032=1219.985,90.748,-47.659,-178.622,5.614,148.574
C07033=1219.989,90.499,-47.641,-178.625,5.614,148.575
C07034=1219.994,90.249,-47.623,-178.627,5.613,148.575
C07035=1219.999,90.000,-47.605,-178.629,5.612,148.576
C07036=1220.004,89.750,-47.586,-178.633,5.611,148.576
C07037=1220.009,89.501,-47.568,-178.635,5.610,148.577
C07038=1220.014,89.252,-47.550,-178.637,5.609,148.578
C07039=1220.019,89.003,-47.532,-178.640,5.609,148.578
C07040=1220.024,88.754,-47.513,-178.642,5.608,148.579
C07041=1220.028,88.504,-47.495,-178.645,5.607,148.579
C07042=1220.033,88.255,-47.477,-178.648,5.606,148.580
C07043=1220.038,88.006,-47.459,-178.650,5.605,148.580
C07044=1220.043,87.757,-47.441,-178.653,5.604,148.581
C07045=1220.048,87.507,-47.423,-178.655,5.603,148.582
C07046=1220.053,87.258,-47.404,-178.657,5.603,148.582
C07047=1220.058,87.008,-47.386,-178.660,5.602,148.583
C07048=1220.062,86.759,-47.368,-178.663,5.601,148.583
C07049=1220.067,86.510,-47.350,-178.666,5.600,148.584
C07050=1220.072,86.261,-47.332,-178.668,5.599,148.584
C07051=1220.077,86.011,-47.314,-178.671,5.598,148.585
C07052=1220.082,85.762,-47.296,-178.673,5.598,148.586
C07053=1220.087,85.513,-47.278,-178.675,5.597,148.586
C07054=1220.091,85.263,-47.260,-178.678,5.595,148.587
C07055=1220.096,85.014,-47.242,-178.681,5.595,148.587
C07056=1220.101,84.765,-47.224,-178.683,5.594,148.588
C07057=1220.106,84.516,-47.206,-178.686,5.593,148.589
C07058=1220.111,84.266,-47.188,-178.688,5.593,148.589
C07059=1220.116,84.017,-47.171,-178.691,5.592,148.590
C07060=1220.121,83.767,-47.153,-178.693,5.591,148.590
C07061=1220.126,83.518,-47.135,-178.696,5.590,148.591
C07062=1220.130,83.268,-47.116,-178.699,5.589,148.592
C07063=1220.135,83.019,-47.098,-178.701,5.588,148.592
C07064=1220.140,82.770,-47.080,-178.704,5.588,148.593
C07065=1220.145,82.521,-47.062,-178.706,5.587,148.593
C07066=1220.150,82.272,-47.044,-178.709,5.587,148.594
C07067=1220.155,82.022,-47.027,-178.711,5.586,148.594
C07068=1220.160,81.754,-47.008,-178.714,5.584,148.595
C07069=1220.165,81.485,-46.988,-178.717,5.584,148.596
C07070=1220.170,81.217,-46.969,-178.720,5.583,148.596
C07071=1220.176,80.948,-46.950,-178.723,5.582,148.597
C07072=1220.181,80.699,-46.932,-178.725,5.581,148.598
C07073=1220.186,80.450,-46.914,-178.728,5.580,148.598
C07074=1220.191,80.201,-46.896,-178.730,5.580,148.599
C07075=1220.195,79.952,-46.879,-178.733,5.579,148.599
C07076=1220.200,79.702,-46.862,-178.735,5.578,148.600
C07077=1220.205,79.453,-46.844,-178.738,5.577,148.601
C07078=1220.210,79.204,-46.826,-178.741,5.576,148.601
C07079=1220.215,78.955,-46.808,-178.743,5.575,148.602
C07080=1220.220,78.705,-46.790,-178.746,5.574,148.602
C07081=1220.225,78.456,-46.772,-178.748,5.574,148.603
C07082=1220.230,78.206,-46.754,-178.751,5.573,148.604
C07083=1220.234,77.957,-46.738,-178.753,5.573,148.604
C07084=1220.239,77.708,-46.720,-178.756,5.572,148.605
C07085=1220.244,77.459,-46.702,-178.758,5.571,148.605
C07086=1220.249,77.209,-46.684,-178.761,5.571,148.606
C07087=1220.254,76.960,-46.667,-178.764,5.569,148.607
C07088=1220.259,76.710,-46.649,-178.766,5.568,148.607
C07089=1220.264,76.461,-46.632,-178.769,5.568,148.608
C07090=1220.268,76.212,-46.614,-178.771,5.567,148.608
C07091=1220.273,75.963,-46.596,-178.774,5.567,148.609
C07092=1220.279,75.713,-46.579,-178.776,5.566,148.609
C07093=1220.284,75.464,-46.561,-178.779,5.565,148.610
C07094=1220.288,75.215,-46.543,-178.781,5.564,148.611
C07095=1220.293,74.965,-46.526,-178.784,5.564,148.611
C07096=1220.298,74.716,-46.508,-178.786,5.563,148.612
C07097=1220.303,74.466,-46.491,-178.789,5.562,148.612
C07098=1220.307,74.217,-46.473,-178.792,5.561,148.613
C07099=1220.312,73.967,-46.456,-178.794,5.560,148.614
C07100=1220.317,73.718,-46.438,-178.797,5.559,148.614
C07101=1220.322,73.469,-46.420,-178.799,5.559,148.615
C07102=1220.327,73.219,-46.403,-178.802,5.558,148.616
C07103=1220.332,72.970,-46.386,-178.804,5.557,148.616
C07104=1220.337,72.721,-46.368,-178.807,5.557,148.617
C07105=1220.341,72.472,-46.351,-178.809,5.556,148.617
C07106=1220.346,72.222,-46.334,-178.812,5.556,148.618
C07107=1220.351,71.973,-46.316,-178.815,5.555,148.619
C07108=1220.357,71.724,-46.299,-178.817,5.553,148.619
C07109=1220.361,71.475,-46.281,-178.820,5.553,148.620
C07110=1220.366,71.225,-46.264,-178.823,5.552,148.620
C07111=1220.372,70.975,-46.247,-178.825,5.552,148.621
C07112=1220.376,70.726,-46.229,-178.827,5.551,148.621
C07113=1220.381,70.476,-46.212,-178.830,5.550,148.622
C07114=1220.386,70.227,-46.194,-178.833,5.549,148.623
C07115=1220.390,69.978,-46.178,-178.835,5.549,148.623
C07116=1220.395,69.729,-46.160,-178.837,5.548,148.624
C07117=1220.401,69.479,-46.142,-178.840,5.547,148.625
C07118=1220.406,69.230,-46.126,-178.843,5.547,148.625
C07119=1220.411,68.981,-46.108,-178.845,5.546,148.626
C07120=1220.415,68.731,-46.091,-178.847,5.545,148.626
C07121=1220.420,68.482,-46.073,-178.851,5.544,148.627
C07122=1220.425,68.232,-46.056,-178.853,5.543,148.628
C07123=1220.430,67.983,-46.039,-178.856,5.543,148.628
C07124=1220.435,67.734,-46.021,-178.859,5.542,148.629
C07125=1220.439,67.484,-46.005,-178.861,5.541,148.629
C07126=1220.445,67.235,-45.988,-178.863,5.541,148.630
C07127=1220.450,66.986,-45.970,-178.866,5.540,148.631
C07128=1220.454,66.737,-45.953,-178.869,5.540,148.631
C07129=1220.459,66.487,-45.936,-178.871,5.539,148.632
C07130=1220.464,66.238,-45.919,-178.873,5.538,148.632
C07131=1220.469,65.988,-45.901,-178.876,5.537,148.633
C07132=1220.474,65.739,-45.885,-178.879,5.537,148.634
C07133=1220.479,65.490,-45.868,-178.881,5.536,148.634
C07134=1220.483,65.241,-45.850,-178.883,5.535,148.635
C07135=1220.489,64.991,-45.833,-178.886,5.535,148.636
C07136=1220.493,64.741,-45.816,-178.889,5.534,148.636
C07137=1220.498,64.492,-45.799,-178.891,5.534,148.637
C07138=1220.503,64.243,-45.782,-178.893,5.533,148.637
C07139=1220.508,63.994,-45.765,-178.897,5.531,148.638
C07140=1220.513,63.744,-45.748,-178.899,5.531,148.639
C07141=1220.518,63.494,-45.731,-178.902,5.530,148.639
C07142=1220.522,63.245,-45.714,-178.905,5.530,148.640
C07143=1220.528,62.996,-45.697,-178.907,5.529,148.640
C07144=1220.532,62.747,-45.680,-178.909,5.528,148.641
C07145=1220.538,62.497,-45.663,-178.912,5.528,148.642
C07146=1220.542,62.248,-45.646,-178.915,5.527,148.642
C07147=1220.548,61.999,-45.629,-178.917,5.526,148.643
C07148=1220.552,61.749,-45.612,-178.919,5.526,148.643
C07149=1220.558,61.499,-45.595,-178.922,5.525,148.644
C07150=1220.562,61.250,-45.578,-178.925,5.524,148.645
C07151=1220.568,61.001,-45.561,-178.927,5.524,148.645
C07152=1220.572,60.752,-45.544,-178.930,5.523,148.646
C07153=1220.577,60.502,-45.528,-178.932,5.522,148.647
C07154=1220.582,60.253,-45.510,-178.935,5.522,148.647
C07155=1220.587,60.004,-45.494,-178.937,5.521,148.648
C07156=1220.592,59.754,-45.477,-178.940,5.521,148.649
C07157=1220.597,59.504,-45.460,-178.943,5.520,148.649
C07158=1220.601,59.255,-45.443,-178.945,5.519,148.650
C07159=1220.607,59.006,-45.427,-178.947,5.519,148.650
C07160=1220.611,58.756,-45.410,-178.950,5.518,148.651
C07161=1220.617,58.507,-45.393,-178.953,5.517,148.652
C07162=1220.621,58.257,-45.376,-178.955,5.517,148.652
C07163=1220.626,58.008,-45.360,-178.957,5.516,148.653
C07164=1220.631,57.759,-45.342,-178.960,5.515,148.653
C07165=1220.636,57.509,-45.326,-178.963,5.515,148.654
C07166=1220.641,57.260,-45.309,-178.965,5.514,148.655
C07167=1220.646,57.010,-45.292,-178.968,5.514,148.655
C07168=1220.651,56.761,-45.275,-178.971,5.513,148.656
C07169=1220.656,56.512,-45.259,-178.973,5.512,148.657
C07170=1220.661,56.262,-45.242,-178.975,5.512,148.657
C07171=1220.665,56.013,-45.225,-178.978,5.511,148.658
C07172=1220.671,55.745,-45.207,-178.981,5.510,148.659
C07173=1220.676,55.476,-45.189,-178.984,5.509,148.659
C07174=1220.682,55.208,-45.172,-178.986,5.509,148.660
C07175=1220.687,54.939,-45.153,-178.989,5.508,148.661
C07176=1220.692,54.690,-45.137,-178.992,5.507,148.661
C07177=1220.697,54.441,-45.120,-178.994,5.507,148.662
C07178=1220.701,54.191,-45.103,-178.997,5.506,148.663
C07179=1220.707,53.942,-45.087,-178.999,5.505,148.663
C07180=1220.711,53.693,-45.070,-179.002,5.505,148.664
C07181=1220.717,53.443,-45.054,-179.004,5.504,148.664
C07182=1220.721,53.194,-45.038,-179.007,5.504,148.665
C07183=1220.726,52.944,-45.020,-179.010,5.503,148.666
C07184=1220.731,52.695,-45.004,-179.012,5.503,148.666
C07185=1220.736,52.446,-44.987,-179.014,5.502,148.667
C07186=1220.740,52.196,-44.971,-179.017,5.501,148.667
C07187=1220.747,51.946,-44.955,-179.020,5.500,148.668
C07188=1220.751,51.697,-44.938,-179.022,5.500,148.669
C07189=1220.756,51.448,-44.922,-179.025,5.499,148.669
C07190=1220.761,51.199,-44.905,-179.028,5.499,148.670
C07191=1220.765,50.949,-44.888,-179.030,5.498,148.671
C07192=1220.771,50.699,-44.872,-179.032,5.497,148.671
C07193=1220.776,50.450,-44.855,-179.035,5.497,148.672
C07194=1220.781,50.201,-44.839,-179.038,5.496,148.673
C07195=1220.785,49.952,-44.822,-179.040,5.496,148.673
C07196=1220.790,49.702,-44.806,-179.043,5.495,148.674
C07197=1220.795,49.453,-44.790,-179.045,5.494,148.674
C07198=1220.800,49.203,-44.773,-179.048,5.494,148.675
C07199=1220.806,48.954,-44.757,-179.050,5.493,148.676
C07200=1220.810,48.704,-44.741,-179.052,5.493,148.676
C07201=1220.815,48.455,-44.724,-179.055,5.493,148.677
C07202=1220.820,48.205,-44.708,-179.058,5.492,148.678
C07203=1220.825,47.956,-44.692,-179.060,5.491,148.678
C07204=1220.830,47.707,-44.675,-179.063,5.491,148.679
C07205=1220.834,47.457,-44.659,-179.065,5.490,148.679
C07206=1220.840,47.208,-44.643,-179.068,5.490,148.680
C07207=1220.845,46.958,-44.626,-179.070,5.489,148.681
C07208=1220.850,46.709,-44.610,-179.073,5.488,148.681
C07209=1220.855,46.459,-44.594,-179.076,5.488,148.682
C07210=1220.860,46.211,-44.577,-179.078,5.487,148.683
C07211=1220.864,45.960,-44.561,-179.080,5.486,148.683
C07212=1220.869,45.712,-44.545,-179.083,5.486,148.684
C07213=1220.874,45.462,-44.529,-179.086,5.485,148.685
C07214=1220.879,45.212,-44.512,-179.088,5.485,148.685
C07215=1220.884,44.963,-44.497,-179.091,5.484,148.686
C07216=1220.889,44.713,-44.480,-179.094,5.484,148.687
C07217=1220.894,44.464,-44.464,-179.096,5.483,148.687
C07218=1220.898,44.214,-44.448,-179.098,5.482,148.688
C07219=1220.904,43.966,-44.432,-179.101,5.482,148.688
C07220=1220.908,43.715,-44.416,-179.104,5.481,148.689
C07221=1220.913,43.467,-44.399,-179.106,5.481,148.690
C07222=1220.919,43.217,-44.384,-179.109,5.480,148.690
C07223=1220.923,42.968,-44.367,-179.111,5.480,148.691
C07224=1220.929,42.718,-44.351,-179.113,5.479,148.692
C07225=1220.933,42.469,-44.335,-179.116,5.479,148.692
C07226=1220.939,42.220,-44.319,-179.119,5.478,148.693
C07227=1220.943,41.970,-44.303,-179.121,5.478,148.694
C07228=1220.948,41.721,-44.287,-179.124,5.477,148.694
C07229=1220.953,41.471,-44.270,-179.126,5.477,148.695
C07230=1220.958,41.222,-44.255,-179.129,5.476,148.696
C07231=1220.963,40.972,-44.239,-179.131,5.475,148.696
C07232=1220.968,40.723,-44.222,-179.134,5.475,148.697
C07233=1220.973,40.473,-44.207,-179.136,5.474,148.697
C07234=1220.978,40.224,-44.190,-179.139,5.473,148.698
C07235=1220.983,39.975,-44.175,-179.142,5.473,148.699
C07236=1220.988,39.724,-44.159,-179.144,5.472,148.699
C07237=1220.993,39.476,-44.142,-179.147,5.472,148.700
C07238=1220.998,39.226,-44.126,-179.149,5.472,148.701
C07239=1221.003,38.977,-44.110,-179.151,5.471,148.701
C07240=1221.009,38.727,-44.095,-179.154,5.471,148.702
C07241=1221.013,38.477,-44.079,-179.157,5.470,148.703
C07242=1221.018,38.228,-44.062,-179.159,5.470,148.703
C07243=1221.023,37.978,-44.046,-179.162,5.469,148.704
C07244=1221.028,37.729,-44.031,-179.164,5.468,148.705
C07245=1221.033,37.481,-44.015,-179.167,5.468,148.705
C07246=1221.038,37.230,-43.999,-179.170,5.467,148.706
C07247=1221.043,36.981,-43.983,-179.172,5.466,148.706
C07248=1221.048,36.732,-43.967,-179.175,5.466,148.707
C07249=1221.053,36.482,-43.951,-179.177,5.465,148.708
C07250=1221.058,36.233,-43.936,-179.179,5.466,148.708
C07251=1221.062,35.983,-43.920,-179.182,5.465,148.709
C07252=1221.067,35.734,-43.904,-179.185,5.464,148.710
C07253=1221.073,35.485,-43.888,-179.187,5.464,148.710
C07254=1221.078,35.235,-43.872,-179.190,5.463,148.711
C07255=1221.083,34.985,-43.857,-179.192,5.463,148.712
C07256=1221.088,34.736,-43.840,-179.195,5.462,148.712
C07257=1221.092,34.487,-43.825,-179.197,5.461,148.713
C07258=1221.098,34.237,-43.810,-179.200,5.461,148.714
C07259=1221.102,33.987,-43.794,-179.203,5.460,148.714
C07260=1221.108,33.738,-43.778,-179.205,5.460,148.715
C07261=1221.113,33.489,-43.762,-179.207,5.460,148.716
C07262=1221.117,33.239,-43.746,-179.210,5.459,148.716
C07263=1221.122,32.990,-43.731,-179.213,5.459,148.717
C07264=1221.128,32.740,-43.715,-179.215,5.458,148.718
C07265=1221.132,32.490,-43.699,-179.217,5.457,148.718
C07266=1221.137,32.241,-43.684,-179.220,5.457,148.719
C07267=1221.142,31.992,-43.668,-179.223,5.456,148.719
C07268=1221.147,31.742,-43.652,-179.225,5.456,148.720
C07269=1221.152,31.493,-43.636,-179.228,5.455,148.721
C07270=1221.157,31.244,-43.621,-179.231,5.455,148.721
C07271=1221.162,30.994,-43.606,-179.233,5.455,148.722
C07272=1221.167,30.744,-43.590,-179.235,5.454,148.723
C07273=1221.173,30.495,-43.574,-179.238,5.454,148.723
C07274=1221.177,30.246,-43.559,-179.240,5.453,148.724
C07275=1221.182,29.996,-43.543,-179.243,5.453,148.725
C07276=1221.188,29.727,-43.526,-179.245,5.452,148.725
C07277=1221.193,29.459,-43.509,-179.248,5.452,148.726
C07278=1221.198,29.191,-43.493,-179.251,5.451,148.727
C07279=1221.204,28.921,-43.477,-179.254,5.451,148.728
C07280=1221.209,28.672,-43.461,-179.256,5.450,148.728
C07281=1221.213,28.422,-43.446,-179.259,5.450,148.729
C07282=1221.219,28.173,-43.430,-179.262,5.449,148.730
C07283=1221.224,27.923,-43.414,-179.264,5.448,148.730
C07284=1221.229,27.674,-43.399,-179.266,5.448,148.731
C07285=1221.233,27.424,-43.384,-179.269,5.448,148.731
C07286=1221.239,27.175,-43.368,-179.271,5.447,148.732
C07287=1221.243,26.926,-43.353,-179.274,5.447,148.733
C07288=1221.249,26.676,-43.337,-179.277,5.446,148.733
C07289=1221.254,26.426,-43.321,-179.279,5.446,148.734
C07290=1221.258,26.177,-43.306,-179.282,5.445,148.735
C07291=1221.264,25.928,-43.291,-179.284,5.445,148.735
C07292=1221.268,25.679,-43.276,-179.287,5.445,148.736
C07293=1221.274,25.429,-43.260,-179.289,5.444,148.737
C07294=1221.278,25.179,-43.244,-179.291,5.444,148.737
